	VAR robtarget Openhole_2075 := [[461.97, -18.21, 181.08], [0.041173, 0.705907, 0.7057, -0.044582], [0,0,0,0], [9E9, 9E9, 9E9, 9E9, 9E9, 9E9]];
	VAR robtarget Openhole_2076 := [[462.15, -19.58, 181.25], [0.046371, 0.705585, 0.705943, -0.04055], [0,0,0,0], [9E9, 9E9, 9E9, 9E9, 9E9, 9E9]];
	VAR robtarget Openhole_2077 := [[462.64, -19.54, 181.25], [0.047892, 0.705483, 0.705837, -0.04236], [0,0,0,0], [9E9, 9E9, 9E9, 9E9, 9E9, 9E9]];
	VAR robtarget Openhole_2078 := [[463.64, -19.43, 181.24], [0.050847, 0.705276, 0.705606, -0.046042], [0,0,0,0], [9E9, 9E9, 9E9, 9E9, 9E9, 9E9]];
	VAR robtarget Openhole_2079 := [[464.14, -19.42, 181.24], [0.052483, 0.705156, 0.705494, -0.047735], [0,0,0,0], [9E9, 9E9, 9E9, 9E9, 9E9, 9E9]];
	VAR robtarget Openhole_2080 := [[464.64, -19.38, 181.23], [0.054002, 0.705042, 0.70537, -0.049529], [0,0,0,0], [9E9, 9E9, 9E9, 9E9, 9E9, 9E9]];
	VAR robtarget Openhole_2081 := [[465.63, -19.33, 181.23], [0.05712, 0.704796, 0.705115, -0.053034], [0,0,0,0], [9E9, 9E9, 9E9, 9E9, 9E9, 9E9]];
	VAR robtarget Openhole_2082 := [[466.13, -19.31, 181.23], [0.058717, 0.704665, 0.704985, -0.054743], [0,0,0,0], [9E9, 9E9, 9E9, 9E9, 9E9, 9E9]];
	VAR robtarget Openhole_2083 := [[466.63, -19.31, 181.23], [0.060351, 0.704527, 0.704853, -0.056412], [0,0,0,0], [9E9, 9E9, 9E9, 9E9, 9E9, 9E9]];
	VAR robtarget Openhole_2084 := [[469.13, -19.24, 181.22], [0.068296, 0.703801, 0.704124, -0.064882], [0,0,0,0], [9E9, 9E9, 9E9, 9E9, 9E9, 9E9]];
	VAR robtarget Openhole_2085 := [[469.63, -19.24, 181.22], [0.069931, 0.70364, 0.703972, -0.066512], [0,0,0,0], [9E9, 9E9, 9E9, 9E9, 9E9, 9E9]];
	VAR robtarget Openhole_2086 := [[470.13, -19.24, 181.22], [0.071554, 0.703477, 0.703815, -0.068148], [0,0,0,0], [9E9, 9E9, 9E9, 9E9, 9E9, 9E9]];
	VAR robtarget Openhole_2087 := [[470.63, -19.24, 181.23], [0.073176, 0.70331, 0.703656, -0.069778], [0,0,0,0], [9E9, 9E9, 9E9, 9E9, 9E9, 9E9]];
	VAR robtarget Openhole_2088 := [[490.13, -19.56, 181.39], [0.134065, 0.694281, 0.695212, -0.129154], [0,0,0,0], [9E9, 9E9, 9E9, 9E9, 9E9, 9E9]];
	VAR robtarget Openhole_2089 := [[490.63, -19.56, 181.39], [0.135501, 0.694002, 0.69494, -0.130609], [0,0,0,0], [9E9, 9E9, 9E9, 9E9, 9E9, 9E9]];
	VAR robtarget Openhole_2090 := [[499.63, -19.4, 181.36], [0.159952, 0.688778, 0.689613, -0.156314], [0,0,0,0], [9E9, 9E9, 9E9, 9E9, 9E9, 9E9]];
	VAR robtarget Openhole_2091 := [[504.35, -19.19, 181.27], [0.171684, 0.685948, 0.686508, -0.169431], [0,0,0,0], [9E9, 9E9, 9E9, 9E9, 9E9, 9E9]];
	VAR robtarget Openhole_2092 := [[536.35, -19.19, 181.19], [0.183051, 0.683002, 0.683002, -0.183051], [0,0,0,0], [9E9, 9E9, 9E9, 9E9, 9E9, 9E9]];
	VAR robtarget Openhole_2093 := [[536.35, -19.88, 181.59], [0.183051, 0.683002, 0.683002, -0.183051], [0,0,0,0], [9E9, 9E9, 9E9, 9E9, 9E9, 9E9]];
	VAR robtarget Openhole_2094 := [[509.35, -19.88, 181.68], [0.183051, 0.683002, 0.683002, -0.183051], [0,0,0,0], [9E9, 9E9, 9E9, 9E9, 9E9, 9E9]];
	VAR robtarget Openhole_2095 := [[504.35, -19.88, 181.64], [0.173716, 0.685436, 0.687007, -0.167394], [0,0,0,0], [9E9, 9E9, 9E9, 9E9, 9E9, 9E9]];
	VAR robtarget Openhole_2096 := [[495.85, -20.21, 181.71], [0.152146, 0.690544, 0.692397, -0.14348], [0,0,0,0], [9E9, 9E9, 9E9, 9E9, 9E9, 9E9]];
	VAR robtarget Openhole_2097 := [[489.35, -20.27, 181.66], [0.134036, 0.694287, 0.696036, -0.124637], [0,0,0,0], [9E9, 9E9, 9E9, 9E9, 9E9, 9E9]];
	VAR robtarget Openhole_2098 := [[488.85, -20.27, 181.65], [0.132589, 0.694565, 0.696297, -0.123167], [0,0,0,0], [9E9, 9E9, 9E9, 9E9, 9E9, 9E9]];
	VAR robtarget Openhole_2099 := [[474.85, -20.03, 181.43], [0.089308, 0.701444, 0.702476, -0.080793], [0,0,0,0], [9E9, 9E9, 9E9, 9E9, 9E9, 9E9]];
	VAR robtarget Openhole_2100 := [[470.86, -19.93, 181.37], [0.076174, 0.702992, 0.703809, -0.068212], [0,0,0,0], [9E9, 9E9, 9E9, 9E9, 9E9, 9E9]];
	VAR robtarget Openhole_2101 := [[473.3, -13.93, 180.01], [0.064302, 0.704177, 0.700574, -0.095897], [0,0,0,0], [9E9, 9E9, 9E9, 9E9, 9E9, 9E9]];
	VAR robtarget Openhole_2102 := [[474.29, -13.82, 179.93], [0.067149, 0.703911, 0.700086, -0.099395], [0,0,0,0], [9E9, 9E9, 9E9, 9E9, 9E9, 9E9]];
	VAR robtarget Openhole_2103 := [[479.28, -13.55, 179.6], [0.082192, 0.702314, 0.697567, -0.11576], [0,0,0,0], [9E9, 9E9, 9E9, 9E9, 9E9, 9E9]];
	VAR robtarget Openhole_2104 := [[482.27, -13.53, 179.44], [0.091487, 0.701163, 0.695983, -0.12493], [0,0,0,0], [9E9, 9E9, 9E9, 9E9, 9E9, 9E9]];
	VAR robtarget Openhole_2105 := [[482.77, -13.53, 179.41], [0.093043, 0.700959, 0.695714, -0.12642], [0,0,0,0], [9E9, 9E9, 9E9, 9E9, 9E9, 9E9]];
	VAR robtarget Openhole_2106 := [[494.76, -13.69, 178.85], [0.129253, 0.695193, 0.688701, -0.160282], [0,0,0,0], [9E9, 9E9, 9E9, 9E9, 9E9, 9E9]];
	VAR robtarget Openhole_2107 := [[495.25, -13.69, 178.82], [0.130674, 0.694928, 0.688382, -0.161647], [0,0,0,0], [9E9, 9E9, 9E9, 9E9, 9E9, 9E9]];
	VAR robtarget Openhole_2108 := [[501.74, -13.52, 178.4], [0.148158, 0.691411, 0.683992, -0.179317], [0,0,0,0], [9E9, 9E9, 9E9, 9E9, 9E9, 9E9]];
	VAR robtarget Openhole_2109 := [[504.34, -13.35, 178.17], [0.154616, 0.689996, 0.682093, -0.186411], [0,0,0,0], [9E9, 9E9, 9E9, 9E9, 9E9, 9E9]];
	VAR robtarget Openhole_2110 := [[509.34, -13.35, 177.9], [0.183051, 0.683002, 0.683002, -0.183051], [0,0,0,0], [9E9, 9E9, 9E9, 9E9, 9E9, 9E9]];
	VAR robtarget Openhole_2111 := [[536.34, -13.35, 177.82], [0.183051, 0.683002, 0.683002, -0.183051], [0,0,0,0], [9E9, 9E9, 9E9, 9E9, 9E9, 9E9]];
	VAR robtarget Openhole_2112 := [[536.33, -11.35, 176.66], [0.183051, 0.683002, 0.683002, -0.183051], [0,0,0,0], [9E9, 9E9, 9E9, 9E9, 9E9, 9E9]];
	VAR robtarget Openhole_2113 := [[509.33, -11.35, 176.75], [0.183051, 0.683002, 0.683002, -0.183051], [0,0,0,0], [9E9, 9E9, 9E9, 9E9, 9E9, 9E9]];
	VAR robtarget Openhole_2114 := [[504.33, -11.35, 177.12], [0.148768, 0.69128, 0.68049, -0.192181], [0,0,0,0], [9E9, 9E9, 9E9, 9E9, 9E9, 9E9]];
	VAR robtarget Openhole_2115 := [[503.51, -11.37, 177.19], [0.146636, 0.691735, 0.681083, -0.190069], [0,0,0,0], [9E9, 9E9, 9E9, 9E9, 9E9, 9E9]];
	VAR robtarget Openhole_2116 := [[498.54, -11.56, 177.65], [0.133524, 0.694386, 0.684651, -0.176787], [0,0,0,0], [9E9, 9E9, 9E9, 9E9, 9E9, 9E9]];
	VAR robtarget Openhole_2117 := [[497.54, -11.57, 177.72], [0.130734, 0.694916, 0.685326, -0.174149], [0,0,0,0], [9E9, 9E9, 9E9, 9E9, 9E9, 9E9]];
	VAR robtarget Openhole_2118 := [[497.04, -11.57, 177.76], [0.129318, 0.695181, 0.685659, -0.172833], [0,0,0,0], [9E9, 9E9, 9E9, 9E9, 9E9, 9E9]];
	VAR robtarget Openhole_2119 := [[482.58, -11.27, 178.7], [0.085227, 0.701952, 0.694483, -0.133017], [0,0,0,0], [9E9, 9E9, 9E9, 9E9, 9E9, 9E9]];
	VAR robtarget Openhole_2120 := [[482.08, -11.28, 178.74], [0.083674, 0.702139, 0.694767, -0.131526], [0,0,0,0], [9E9, 9E9, 9E9, 9E9, 9E9, 9E9]];
	VAR robtarget Openhole_2121 := [[477.1, -11.44, 179.15], [0.068397, 0.703791, 0.697543, -0.115903], [0,0,0,0], [9E9, 9E9, 9E9, 9E9, 9E9, 9E9]];
	VAR robtarget Openhole_2122 := [[473.15, -11.89, 179.55], [0.05708, 0.704799, 0.699699, -0.102087], [0,0,0,0], [9E9, 9E9, 9E9, 9E9, 9E9, 9E9]];
	VAR robtarget Openhole_2123 := [[471.68, -12.15, 179.7], [0.053121, 0.705109, 0.70048, -0.096583], [0,0,0,0], [9E9, 9E9, 9E9, 9E9, 9E9, 9E9]];
	VAR robtarget Openhole_2124 := [[471.19, -12.25, 179.76], [0.05186, 0.705202, 0.700737, -0.094695], [0,0,0,0], [9E9, 9E9, 9E9, 9E9, 9E9, 9E9]];
	VAR robtarget Openhole_2125 := [[470.71, -12.36, 179.81], [0.050637, 0.705291, 0.700994, -0.092778], [0,0,0,0], [9E9, 9E9, 9E9, 9E9, 9E9, 9E9]];
	VAR robtarget Openhole_2126 := [[469.27, -12.75, 179.98], [0.047173, 0.705531, 0.70175, -0.086871], [0,0,0,0], [9E9, 9E9, 9E9, 9E9, 9E9, 9E9]];
	VAR robtarget Openhole_2127 := [[468.32, -13.04, 180.09], [0.044997, 0.705674, 0.702239, -0.082831], [0,0,0,0], [9E9, 9E9, 9E9, 9E9, 9E9, 9E9]];
	VAR robtarget Openhole_2128 := [[467.85, -13.2, 180.14], [0.043961, 0.705739, 0.702478, -0.080777], [0,0,0,0], [9E9, 9E9, 9E9, 9E9, 9E9, 9E9]];
	VAR robtarget Openhole_2129 := [[467.38, -13.37, 180.2], [0.042984, 0.705799, 0.702715, -0.078688], [0,0,0,0], [9E9, 9E9, 9E9, 9E9, 9E9, 9E9]];
	VAR robtarget Openhole_2130 := [[466.46, -13.74, 180.31], [0.04115, 0.705908, 0.703177, -0.074444], [0,0,0,0], [9E9, 9E9, 9E9, 9E9, 9E9, 9E9]];
	VAR robtarget Openhole_2131 := [[466, -13.94, 180.37], [0.040305, 0.705957, 0.703402, -0.072286], [0,0,0,0], [9E9, 9E9, 9E9, 9E9, 9E9, 9E9]];
	VAR robtarget Openhole_2132 := [[465.55, -14.15, 180.42], [0.039502, 0.706003, 0.703623, -0.070106], [0,0,0,0], [9E9, 9E9, 9E9, 9E9, 9E9, 9E9]];
	VAR robtarget Openhole_2133 := [[464.66, -14.6, 180.53], [0.03804, 0.706083, 0.70405, -0.065683], [0,0,0,0], [9E9, 9E9, 9E9, 9E9, 9E9, 9E9]];
	VAR robtarget Openhole_2134 := [[463.79, -15.08, 180.63], [0.036763, 0.70615, 0.704455, -0.061184], [0,0,0,0], [9E9, 9E9, 9E9, 9E9, 9E9, 9E9]];
	VAR robtarget Openhole_2135 := [[462.94, -15.6, 180.73], [0.035643, 0.706208, 0.704836, -0.056628], [0,0,0,0], [9E9, 9E9, 9E9, 9E9, 9E9, 9E9]];
	VAR robtarget Openhole_2136 := [[462.52, -15.87, 180.78], [0.03514, 0.706233, 0.705017, -0.054329], [0,0,0,0], [9E9, 9E9, 9E9, 9E9, 9E9, 9E9]];
	VAR robtarget Openhole_2137 := [[460.89, -17, 180.96], [0.033479, 0.706314, 0.705672, -0.045027], [0,0,0,0], [9E9, 9E9, 9E9, 9E9, 9E9, 9E9]];
	VAR robtarget Openhole_2138 := [[461.06, -13.27, 180.53], [0.021493, 0.70678, 0.704709, -0.058177], [0,0,0,0], [9E9, 9E9, 9E9, 9E9, 9E9, 9E9]];
	VAR robtarget Openhole_2139 := [[460.62, -13.5, 180.58], [0.020785, 0.706801, 0.704891, -0.055928], [0,0,0,0], [9E9, 9E9, 9E9, 9E9, 9E9, 9E9]];
	VAR robtarget Openhole_2140 := [[458.51, -14.82, 180.81], [0.018075, 0.706876, 0.705711, -0.04441], [0,0,0,0], [9E9, 9E9, 9E9, 9E9, 9E9, 9E9]];
	VAR robtarget Openhole_2141 := [[457.68, -15.38, 180.89], [0.017191, 0.706898, 0.705989, -0.039736], [0,0,0,0], [9E9, 9E9, 9E9, 9E9, 9E9, 9E9]];
	VAR robtarget Openhole_2142 := [[456.81, -15.81, 180.95], [0.01568, 0.706933, 0.706224, -0.035314], [0,0,0,0], [9E9, 9E9, 9E9, 9E9, 9E9, 9E9]];
	VAR robtarget Openhole_2143 := [[457.02, -21.12, 181.34], [0.034402, 0.706269, 0.706877, -0.018011], [0,0,0,0], [9E9, 9E9, 9E9, 9E9, 9E9, 9E9]];
	VAR robtarget Openhole_2144 := [[463.92, -21.12, 181.48], [0.057484, 0.704766, 0.7059, -0.041297], [0,0,0,0], [9E9, 9E9, 9E9, 9E9, 9E9, 9E9]];
	VAR robtarget Openhole_2145 := [[469.41, -21.53, 181.67], [0.076804, 0.702923, 0.704714, -0.05812], [0,0,0,0], [9E9, 9E9, 9E9, 9E9, 9E9, 9E9]];
	VAR robtarget Openhole_2146 := [[482.39, -21.87, 182.08], [0.118549, 0.697098, 0.700201, -0.098586], [0,0,0,0], [9E9, 9E9, 9E9, 9E9, 9E9, 9E9]];
	VAR robtarget Openhole_2147 := [[487.39, -21.9, 182.23], [0.133435, 0.694403, 0.697902, -0.113721], [0,0,0,0], [9E9, 9E9, 9E9, 9E9, 9E9, 9E9]];
	VAR robtarget Openhole_2148 := [[487.89, -21.9, 182.25], [0.134884, 0.694123, 0.697657, -0.115218], [0,0,0,0], [9E9, 9E9, 9E9, 9E9, 9E9, 9E9]];
	VAR robtarget Openhole_2149 := [[498.39, -21.73, 182.46], [0.16361, 0.687918, 0.691889, -0.14591], [0,0,0,0], [9E9, 9E9, 9E9, 9E9, 9E9, 9E9]];
	VAR robtarget Openhole_2150 := [[503.38, -21.52, 182.48], [0.176032, 0.684845, 0.688756, -0.160046], [0,0,0,0], [9E9, 9E9, 9E9, 9E9, 9E9, 9E9]];
	VAR robtarget Openhole_2151 := [[504.35, -21.49, 182.49], [0.178402, 0.684232, 0.688137, -0.162688], [0,0,0,0], [9E9, 9E9, 9E9, 9E9, 9E9, 9E9]];
	VAR robtarget Openhole_2152 := [[509.35, -21.49, 182.61], [0.183051, 0.683002, 0.683002, -0.183051], [0,0,0,0], [9E9, 9E9, 9E9, 9E9, 9E9, 9E9]];
	VAR robtarget Openhole_2153 := [[536.24, -21.49, 182.52], [0.183051, 0.683002, 0.683002, -0.183051], [0,0,0,0], [9E9, 9E9, 9E9, 9E9, 9E9, 9E9]];
	VAR robtarget Openhole_2154 := [[536.33, -31.04, 188.04], [0.183051, 0.683002, 0.683002, -0.183051], [0,0,0,0], [9E9, 9E9, 9E9, 9E9, 9E9, 9E9]];
	VAR robtarget Openhole_2155 := [[509.37, -31.04, 188.12], [0.183051, 0.683002, 0.683002, -0.183051], [0,0,0,0], [9E9, 9E9, 9E9, 9E9, 9E9, 9E9]];
	VAR robtarget Openhole_2156 := [[504.38, -31.04, 187.54], [0.205934, 0.676455, 0.694141, -0.134788], [0,0,0,0], [9E9, 9E9, 9E9, 9E9, 9E9, 9E9]];
	VAR robtarget Openhole_2157 := [[486.98, -32.16, 185.94], [0.164078, 0.687807, 0.702555, -0.080102], [0,0,0,0], [9E9, 9E9, 9E9, 9E9, 9E9, 9E9]];
	VAR robtarget Openhole_2158 := [[478.56, -33.01, 185.11], [0.142475, 0.692604, 0.705303, -0.050481], [0,0,0,0], [9E9, 9E9, 9E9, 9E9, 9E9, 9E9]];
	VAR robtarget Openhole_2159 := [[471.67, -34.05, 184.41], [0.124885, 0.695991, 0.706689, -0.024306], [0,0,0,0], [9E9, 9E9, 9E9, 9E9, 9E9, 9E9]];
	VAR robtarget Openhole_2160 := [[465.83, -35.24, 183.75], [0.110356, 0.698442, 0.707106, -0.000639], [0,0,0,0], [9E9, 9E9, 9E9, 9E9, 9E9, 9E9]];
	VAR robtarget Openhole_2161 := [[458.15, -37.22, 182.72], [0.091834, 0.701118, 0.706377, 0.032124], [0,0,0,0], [9E9, 9E9, 9E9, 9E9, 9E9, 9E9]];
	VAR robtarget Openhole_2162 := [[452.92, -38.7, 181.86], [0.079284, 0.702648, 0.704975, 0.054868], [0,0,0,0], [9E9, 9E9, 9E9, 9E9, 9E9, 9E9]];
	VAR robtarget Openhole_2163 := [[457.28, -38.7, 182.68], [0.093765, 0.700862, 0.705976, 0.039977], [0,0,0,0], [9E9, 9E9, 9E9, 9E9, 9E9, 9E9]];
	VAR robtarget Openhole_2164 := [[457.75, -38.56, 182.76], [0.094884, 0.700712, 0.706092, 0.037872], [0,0,0,0], [9E9, 9E9, 9E9, 9E9, 9E9, 9E9]];
	VAR robtarget Openhole_2165 := [[466.4, -36.39, 184.03], [0.115866, 0.697549, 0.707106, 0.001208], [0,0,0,0], [9E9, 9E9, 9E9, 9E9, 9E9, 9E9]];
	VAR robtarget Openhole_2166 := [[473.19, -34.93, 184.83], [0.132384, 0.694604, 0.706609, -0.026523], [0,0,0,0], [9E9, 9E9, 9E9, 9E9, 9E9, 9E9]];
	VAR robtarget Openhole_2167 := [[479.58, -33.93, 185.52], [0.148359, 0.691368, 0.705275, -0.050864], [0,0,0,0], [9E9, 9E9, 9E9, 9E9, 9E9, 9E9]];
	VAR robtarget Openhole_2168 := [[487.99, -33.03, 186.39], [0.169538, 0.686482, 0.702507, -0.080521], [0,0,0,0], [9E9, 9E9, 9E9, 9E9, 9E9, 9E9]];
	VAR robtarget Openhole_2169 := [[504.38, -31.93, 188.01], [0.208432, 0.675689, 0.69464, -0.132194], [0,0,0,0], [9E9, 9E9, 9E9, 9E9, 9E9, 9E9]];
	VAR robtarget Openhole_2170 := [[509.37, -31.93, 188.63], [0.183051, 0.683002, 0.683002, -0.183051], [0,0,0,0], [9E9, 9E9, 9E9, 9E9, 9E9, 9E9]];
	VAR robtarget Openhole_2171 := [[536.37, -31.93, 188.55], [0.183051, 0.683002, 0.683002, -0.183051], [0,0,0,0], [9E9, 9E9, 9E9, 9E9, 9E9, 9E9]];
	VAR robtarget Openhole_2172 := [[536.37, -32.81, 189.06], [0.183051, 0.683002, 0.683002, -0.183051], [0,0,0,0], [9E9, 9E9, 9E9, 9E9, 9E9, 9E9]];
	VAR robtarget Openhole_2173 := [[524.37, -32.81, 189.09], [0.183051, 0.683002, 0.683002, -0.183051], [0,0,0,0], [9E9, 9E9, 9E9, 9E9, 9E9, 9E9]];
	VAR robtarget Openhole_2174 := [[509.37, -32.81, 189.14], [0.183051, 0.683002, 0.683002, -0.183051], [0,0,0,0], [9E9, 9E9, 9E9, 9E9, 9E9, 9E9]];
	VAR robtarget Openhole_2175 := [[504.38, -32.81, 188.48], [0.210931, 0.674914, 0.695127, -0.12961], [0,0,0,0], [9E9, 9E9, 9E9, 9E9, 9E9, 9E9]];
	VAR robtarget Openhole_2176 := [[488.99, -33.88, 186.85], [0.17487, 0.685143, 0.702451, -0.081013], [0,0,0,0], [9E9, 9E9, 9E9, 9E9, 9E9, 9E9]];
	VAR robtarget Openhole_2177 := [[481.09, -34.74, 185.98], [0.155283, 0.689846, 0.705104, -0.053183], [0,0,0,0], [9E9, 9E9, 9E9, 9E9, 9E9, 9E9]];
	VAR robtarget Openhole_2178 := [[474.71, -35.76, 185.26], [0.139596, 0.69319, 0.706515, -0.028917], [0,0,0,0], [9E9, 9E9, 9E9, 9E9, 9E9, 9E9]];
	VAR robtarget Openhole_2179 := [[467.43, -37.31, 184.36], [0.122079, 0.696489, 0.707106, 0.000696], [0,0,0,0], [9E9, 9E9, 9E9, 9E9, 9E9, 9E9]];
	VAR robtarget Openhole_2180 := [[462.62, -38.48, 183.66], [0.110468, 0.698425, 0.706797, 0.020931], [0,0,0,0], [9E9, 9E9, 9E9, 9E9, 9E9, 9E9]];
	VAR robtarget Openhole_2181 := [[462.13, -38.7, 183.6], [0.109631, 0.698556, 0.706722, 0.023316], [0,0,0,0], [9E9, 9E9, 9E9, 9E9, 9E9, 9E9]];
	VAR robtarget Openhole_2182 := [[466.52, -38.7, 184.43], [0.123628, 0.696216, 0.707058, 0.00831], [0,0,0,0], [9E9, 9E9, 9E9, 9E9, 9E9, 9E9]];
	VAR robtarget Openhole_2183 := [[467, -38.47, 184.48], [0.124426, 0.696073, 0.707082, 0.00591], [0,0,0,0], [9E9, 9E9, 9E9, 9E9, 9E9, 9E9]];
	VAR robtarget Openhole_2184 := [[474.26, -36.86, 185.46], [0.141738, 0.692756, 0.706704, -0.023852], [0,0,0,0], [9E9, 9E9, 9E9, 9E9, 9E9, 9E9]];
	VAR robtarget Openhole_2185 := [[481.12, -35.71, 186.28], [0.158391, 0.689139, 0.705324, -0.050174], [0,0,0,0], [9E9, 9E9, 9E9, 9E9, 9E9, 9E9]];
	VAR robtarget Openhole_2186 := [[489.01, -34.8, 187.2], [0.177697, 0.684415, 0.702769, -0.078203], [0,0,0,0], [9E9, 9E9, 9E9, 9E9, 9E9, 9E9]];
	VAR robtarget Openhole_2187 := [[501.89, -33.86, 188.68], [0.207948, 0.675838, 0.696929, -0.119541], [0,0,0,0], [9E9, 9E9, 9E9, 9E9, 9E9, 9E9]];
	VAR robtarget Openhole_2188 := [[504.38, -33.69, 188.95], [0.213421, 0.67413, 0.695603, -0.127028], [0,0,0,0], [9E9, 9E9, 9E9, 9E9, 9E9, 9E9]];
	VAR robtarget Openhole_2189 := [[509.37, -33.69, 189.65], [0.183051, 0.683002, 0.683002, -0.183051], [0,0,0,0], [9E9, 9E9, 9E9, 9E9, 9E9, 9E9]];
	VAR robtarget Openhole_2190 := [[536.37, -33.69, 189.57], [0.183051, 0.683002, 0.683002, -0.183051], [0,0,0,0], [9E9, 9E9, 9E9, 9E9, 9E9, 9E9]];
	VAR robtarget Openhole_2191 := [[536.37, -34.58, 190.08], [0.183051, 0.683002, 0.683002, -0.183051], [0,0,0,0], [9E9, 9E9, 9E9, 9E9, 9E9, 9E9]];
	VAR robtarget Openhole_2192 := [[509.37, -34.58, 190.16], [0.183051, 0.683002, 0.683002, -0.183051], [0,0,0,0], [9E9, 9E9, 9E9, 9E9, 9E9, 9E9]];
	VAR robtarget Openhole_2193 := [[504.37, -34.58, 189.41], [0.2159, 0.67334, 0.696071, -0.124442], [0,0,0,0], [9E9, 9E9, 9E9, 9E9, 9E9, 9E9]];
	VAR robtarget Openhole_2194 := [[490.51, -35.57, 187.73], [0.184036, 0.682738, 0.702511, -0.080486], [0,0,0,0], [9E9, 9E9, 9E9, 9E9, 9E9, 9E9]];
	VAR robtarget Openhole_2195 := [[482.13, -36.52, 186.7], [0.163758, 0.687883, 0.705271, -0.050922], [0,0,0,0], [9E9, 9E9, 9E9, 9E9, 9E9, 9E9]];
	VAR robtarget Openhole_2196 := [[475.27, -37.64, 185.82], [0.147219, 0.691611, 0.706674, -0.024743], [0,0,0,0], [9E9, 9E9, 9E9, 9E9, 9E9, 9E9]];
	VAR robtarget Openhole_2197 := [[470.91, -38.55, 185.23], [0.136836, 0.693741, 0.707071, -0.007115], [0,0,0,0], [9E9, 9E9, 9E9, 9E9, 9E9, 9E9]];
	VAR robtarget Openhole_2198 := [[470.42, -38.7, 185.17], [0.135813, 0.693942, 0.707089, -0.004993], [0,0,0,0], [9E9, 9E9, 9E9, 9E9, 9E9, 9E9]];
	VAR robtarget Openhole_2199 := [[474.82, -38.7, 186], [0.149173, 0.691193, 0.706828, -0.019841], [0,0,0,0], [9E9, 9E9, 9E9, 9E9, 9E9, 9E9]];
	VAR robtarget Openhole_2200 := [[475.31, -38.59, 186.07], [0.150274, 0.690954, 0.706769, -0.021839], [0,0,0,0], [9E9, 9E9, 9E9, 9E9, 9E9, 9E9]];
	VAR robtarget Openhole_2201 := [[482.64, -37.38, 187.06], [0.167864, 0.686893, 0.705345, -0.049885], [0,0,0,0], [9E9, 9E9, 9E9, 9E9, 9E9, 9E9]];
	VAR robtarget Openhole_2202 := [[491.02, -36.43, 188.16], [0.187921, 0.681679, 0.70263, -0.07944], [0,0,0,0], [9E9, 9E9, 9E9, 9E9, 9E9, 9E9]];
	VAR robtarget Openhole_2203 := [[502.39, -35.58, 189.63], [0.214044, 0.673933, 0.697545, -0.115895], [0,0,0,0], [9E9, 9E9, 9E9, 9E9, 9E9, 9E9]];
	VAR robtarget Openhole_2204 := [[504.37, -35.46, 189.88], [0.218376, 0.672541, 0.696526, -0.121866], [0,0,0,0], [9E9, 9E9, 9E9, 9E9, 9E9, 9E9]];
	VAR robtarget Openhole_2205 := [[504.37, -35.46, 189.88], [0.21838, 0.67254, 0.696525, -0.121873], [0,0,0,0], [9E9, 9E9, 9E9, 9E9, 9E9, 9E9]];
	VAR robtarget Openhole_2206 := [[509.38, -35.46, 190.67], [0.183051, 0.683002, 0.683002, -0.183051], [0,0,0,0], [9E9, 9E9, 9E9, 9E9, 9E9, 9E9]];
	VAR robtarget Openhole_2207 := [[536.38, -35.46, 190.59], [0.183051, 0.683002, 0.683002, -0.183051], [0,0,0,0], [9E9, 9E9, 9E9, 9E9, 9E9, 9E9]];
	VAR robtarget Openhole_2208 := [[536.38, -36.35, 191.1], [0.183051, 0.683002, 0.683002, -0.183051], [0,0,0,0], [9E9, 9E9, 9E9, 9E9, 9E9, 9E9]];
	VAR robtarget Openhole_2209 := [[509.38, -36.35, 191.18], [0.183051, 0.683002, 0.683002, -0.183051], [0,0,0,0], [9E9, 9E9, 9E9, 9E9, 9E9, 9E9]];
	VAR robtarget Openhole_2210 := [[504.37, -36.35, 190.35], [0.220853, 0.671732, 0.696969, -0.119308], [0,0,0,0], [9E9, 9E9, 9E9, 9E9, 9E9, 9E9]];
	VAR robtarget Openhole_2211 := [[504.37, -36.35, 190.35], [0.220841, 0.671736, 0.696972, -0.119291], [0,0,0,0], [9E9, 9E9, 9E9, 9E9, 9E9, 9E9]];
	VAR robtarget Openhole_2212 := [[503.87, -36.37, 190.28], [0.219768, 0.672088, 0.697224, -0.117808], [0,0,0,0], [9E9, 9E9, 9E9, 9E9, 9E9, 9E9]];
	VAR robtarget Openhole_2213 := [[492.02, -37.26, 188.67], [0.193013, 0.680254, 0.702569, -0.079982], [0,0,0,0], [9E9, 9E9, 9E9, 9E9, 9E9, 9E9]];
	VAR robtarget Openhole_2214 := [[483.16, -38.26, 187.44], [0.172017, 0.685865, 0.705422, -0.04878], [0,0,0,0], [9E9, 9E9, 9E9, 9E9, 9E9, 9E9]];
	VAR robtarget Openhole_2215 := [[480.22, -38.7, 187.02], [0.165, 0.687586, 0.706096, -0.037791], [0,0,0,0], [9E9, 9E9, 9E9, 9E9, 9E9, 9E9]];
	VAR robtarget Openhole_2216 := [[389.31, -38.7, 169.82], [-0.12615, 0.695763, 0.665642, 0.238581], [0,0,0,0], [9E9, 9E9, 9E9, 9E9, 9E9, 9E9]];
	VAR robtarget Openhole_2217 := [[361.4, -38.7, 169.91], [-0.183051, 0.683002, 0.683002, 0.183051], [0,0,0,0], [9E9, 9E9, 9E9, 9E9, 9E9, 9E9]];
	VAR robtarget Openhole_2218 := [[362.33, -29.87, 175], [-0.183051, 0.683002, 0.683002, 0.183051], [0,0,0,0], [9E9, 9E9, 9E9, 9E9, 9E9, 9E9]];
	VAR robtarget Openhole_2219 := [[389.33, -29.87, 174.92], [-0.1512, 0.690752, 0.673839, 0.214338], [0,0,0,0], [9E9, 9E9, 9E9, 9E9, 9E9, 9E9]];
	VAR robtarget Openhole_2220 := [[394.33, -29.87, 175.44], [-0.137763, 0.693557, 0.677476, 0.202551], [0,0,0,0], [9E9, 9E9, 9E9, 9E9, 9E9, 9E9]];
	VAR robtarget Openhole_2221 := [[394.88, -29.88, 175.49], [-0.136237, 0.693858, 0.677866, 0.20124], [0,0,0,0], [9E9, 9E9, 9E9, 9E9, 9E9, 9E9]];
	VAR robtarget Openhole_2222 := [[399.85, -30.07, 175.92], [-0.121699, 0.696555, 0.681266, 0.18941], [0,0,0,0], [9E9, 9E9, 9E9, 9E9, 9E9, 9E9]];
	VAR robtarget Openhole_2223 := [[412.28, -31.06, 176.89], [-0.081421, 0.702403, 0.688984, 0.159062], [0,0,0,0], [9E9, 9E9, 9E9, 9E9, 9E9, 9E9]];
	VAR robtarget Openhole_2224 := [[418.24, -31.27, 177.52], [-0.061858, 0.704396, 0.692601, 0.142491], [0,0,0,0], [9E9, 9E9, 9E9, 9E9, 9E9, 9E9]];
	VAR robtarget Openhole_2225 := [[418.73, -31.27, 177.58], [-0.06026, 0.704534, 0.692902, 0.141019], [0,0,0,0], [9E9, 9E9, 9E9, 9E9, 9E9, 9E9]];
	VAR robtarget Openhole_2226 := [[423.69, -31.07, 178.21], [-0.044741, 0.70569, 0.695888, 0.125456], [0,0,0,0], [9E9, 9E9, 9E9, 9E9, 9E9, 9E9]];
	VAR robtarget Openhole_2227 := [[428.61, -30.5, 178.89], [-0.030265, 0.706459, 0.698762, 0.10831], [0,0,0,0], [9E9, 9E9, 9E9, 9E9, 9E9, 9E9]];
	VAR robtarget Openhole_2228 := [[434.94, -29.34, 179.75], [-0.012795, 0.706991, 0.702086, 0.084111], [0,0,0,0], [9E9, 9E9, 9E9, 9E9, 9E9, 9E9]];
	VAR robtarget Openhole_2229 := [[437.87, -28.76, 180.11], [-0.004847, 0.70709, 0.703374, 0.07256], [0,0,0,0], [9E9, 9E9, 9E9, 9E9, 9E9, 9E9]];
	VAR robtarget Openhole_2230 := [[438.84, -28.58, 180.22], [-0.002113, 0.707104, 0.703759, 0.06873], [0,0,0,0], [9E9, 9E9, 9E9, 9E9, 9E9, 9E9]];
	VAR robtarget Openhole_2231 := [[441.3, -28.17, 180.47], [0.00485, 0.70709, 0.704626, 0.059176], [0,0,0,0], [9E9, 9E9, 9E9, 9E9, 9E9, 9E9]];
	VAR robtarget Openhole_2232 := [[442.28, -28.03, 180.57], [0.007732, 0.707065, 0.704933, 0.055401], [0,0,0,0], [9E9, 9E9, 9E9, 9E9, 9E9, 9E9]];
	VAR robtarget Openhole_2233 := [[445.74, -27.57, 180.88], [0.017944, 0.706879, 0.705846, 0.0422], [0,0,0,0], [9E9, 9E9, 9E9, 9E9, 9E9, 9E9]];
	VAR robtarget Openhole_2234 := [[447.22, -27.43, 181.01], [0.022536, 0.706748, 0.706155, 0.036685], [0,0,0,0], [9E9, 9E9, 9E9, 9E9, 9E9, 9E9]];
	VAR robtarget Openhole_2235 := [[447.72, -27.4, 181.05], [0.02415, 0.706694, 0.706244, 0.034916], [0,0,0,0], [9E9, 9E9, 9E9, 9E9, 9E9, 9E9]];
	VAR robtarget Openhole_2236 := [[448.22, -27.39, 181.09], [0.025802, 0.706636, 0.706328, 0.033182], [0,0,0,0], [9E9, 9E9, 9E9, 9E9, 9E9, 9E9]];
	VAR robtarget Openhole_2237 := [[448.72, -27.39, 181.13], [0.027502, 0.706572, 0.706405, 0.031494], [0,0,0,0], [9E9, 9E9, 9E9, 9E9, 9E9, 9E9]];
	VAR robtarget Openhole_2238 := [[452.7, -27.62, 181.46], [0.041775, 0.705872, 0.706859, 0.018727], [0,0,0,0], [9E9, 9E9, 9E9, 9E9, 9E9, 9E9]];
	VAR robtarget Openhole_2239 := [[454.19, -27.71, 181.59], [0.047103, 0.705536, 0.70697, 0.013931], [0,0,0,0], [9E9, 9E9, 9E9, 9E9, 9E9, 9E9]];
	VAR robtarget Openhole_2240 := [[454.69, -27.73, 181.63], [0.048848, 0.705418, 0.707, 0.012303], [0,0,0,0], [9E9, 9E9, 9E9, 9E9, 9E9, 9E9]];
	VAR robtarget Openhole_2241 := [[455.68, -27.74, 181.71], [0.052246, 0.705174, 0.70705, 0.008952], [0,0,0,0], [9E9, 9E9, 9E9, 9E9, 9E9, 9E9]];
	VAR robtarget Openhole_2242 := [[456.18, -27.73, 181.75], [0.053883, 0.705051, 0.70707, 0.007217], [0,0,0,0], [9E9, 9E9, 9E9, 9E9, 9E9, 9E9]];
	VAR robtarget Openhole_2243 := [[473.12, -27.13, 183.03], [0.107027, 0.69896, 0.705205, -0.051819], [0,0,0,0], [9E9, 9E9, 9E9, 9E9, 9E9, 9E9]];
	VAR robtarget Openhole_2244 := [[498.06, -26.27, 184.58], [0.176241, 0.684791, 0.694806, -0.131317], [0,0,0,0], [9E9, 9E9, 9E9, 9E9, 9E9, 9E9]];
	VAR robtarget Openhole_2245 := [[504.36, -25.98, 184.86], [0.191383, 0.680715, 0.691107, -0.149567], [0,0,0,0], [9E9, 9E9, 9E9, 9E9, 9E9, 9E9]];
	VAR robtarget Openhole_2246 := [[509.36, -25.98, 185.19], [0.183051, 0.683002, 0.683002, -0.183051], [0,0,0,0], [9E9, 9E9, 9E9, 9E9, 9E9, 9E9]];
	VAR robtarget Openhole_2247 := [[536.36, -25.98, 185.11], [0.183051, 0.683002, 0.683002, -0.183051], [0,0,0,0], [9E9, 9E9, 9E9, 9E9, 9E9, 9E9]];
	VAR robtarget Openhole_2248 := [[536.36, -24.92, 184.5], [0.183051, 0.683002, 0.683002, -0.183051], [0,0,0,0], [9E9, 9E9, 9E9, 9E9, 9E9, 9E9]];
	VAR robtarget Openhole_2249 := [[509.36, -24.92, 184.58], [0.183051, 0.683002, 0.683002, -0.183051], [0,0,0,0], [9E9, 9E9, 9E9, 9E9, 9E9, 9E9]];
	VAR robtarget Openhole_2250 := [[504.36, -24.92, 184.3], [0.188332, 0.681565, 0.690431, -0.152662], [0,0,0,0], [9E9, 9E9, 9E9, 9E9, 9E9, 9E9]];
	VAR robtarget Openhole_2251 := [[493.09, -25.36, 183.85], [0.160233, 0.688713, 0.696886, -0.119791], [0,0,0,0], [9E9, 9E9, 9E9, 9E9, 9E9, 9E9]];
	VAR robtarget Openhole_2252 := [[469.64, -25.84, 182.51], [0.091778, 0.701125, 0.705702, -0.044555], [0,0,0,0], [9E9, 9E9, 9E9, 9E9, 9E9, 9E9]];
	VAR robtarget Openhole_2253 := [[467.64, -25.85, 182.38], [0.085401, 0.701931, 0.706092, -0.037869], [0,0,0,0], [9E9, 9E9, 9E9, 9E9, 9E9, 9E9]];
	VAR robtarget Openhole_2254 := [[467.14, -25.85, 182.35], [0.083781, 0.702126, 0.706179, -0.036207], [0,0,0,0], [9E9, 9E9, 9E9, 9E9, 9E9, 9E9]];
	VAR robtarget Openhole_2255 := [[459.66, -25.63, 181.84], [0.058467, 0.704685, 0.70701, -0.011719], [0,0,0,0], [9E9, 9E9, 9E9, 9E9, 9E9, 9E9]];
	VAR robtarget Openhole_2256 := [[455.68, -25.42, 181.57], [0.044398, 0.705712, 0.707106, 0.001113], [0,0,0,0], [9E9, 9E9, 9E9, 9E9, 9E9, 9E9]];
	VAR robtarget Openhole_2257 := [[455.18, -25.38, 181.54], [0.042578, 0.705824, 0.707102, 0.002659], [0,0,0,0], [9E9, 9E9, 9E9, 9E9, 9E9, 9E9]];
	VAR robtarget Openhole_2258 := [[454.68, -25.32, 181.5], [0.040725, 0.705933, 0.707094, 0.004169], [0,0,0,0], [9E9, 9E9, 9E9, 9E9, 9E9, 9E9]];
	VAR robtarget Openhole_2259 := [[454.1, -25.14, 181.46], [0.038116, 0.706079, 0.707085, 0.005549], [0,0,0,0], [9E9, 9E9, 9E9, 9E9, 9E9, 9E9]];
	VAR robtarget Openhole_2260 := [[451.65, -25.14, 181.32], [0.029833, 0.706477, 0.70697, 0.013891], [0,0,0,0], [9E9, 9E9, 9E9, 9E9, 9E9, 9E9]];
	VAR robtarget Openhole_2261 := [[453.07, -23.79, 181.35], [0.030088, 0.706466, 0.707093, 0.004445], [0,0,0,0], [9E9, 9E9, 9E9, 9E9, 9E9, 9E9]];
	VAR robtarget Openhole_2262 := [[455.52, -23.79, 181.46], [0.038358, 0.706066, 0.707096, -0.00389], [0,0,0,0], [9E9, 9E9, 9E9, 9E9, 9E9, 9E9]];
	VAR robtarget Openhole_2263 := [[456.08, -23.86, 181.49], [0.040496, 0.705946, 0.707085, -0.005547], [0,0,0,0], [9E9, 9E9, 9E9, 9E9, 9E9, 9E9]];
	VAR robtarget Openhole_2264 := [[457.08, -23.91, 181.54], [0.044021, 0.705735, 0.707052, -0.00877], [0,0,0,0], [9E9, 9E9, 9E9, 9E9, 9E9, 9E9]];
	VAR robtarget Openhole_2265 := [[458.58, -23.97, 181.62], [0.049247, 0.70539, 0.706975, -0.013649], [0,0,0,0], [9E9, 9E9, 9E9, 9E9, 9E9, 9E9]];
	VAR robtarget Openhole_2266 := [[465.04, -24.53, 182.01], [0.072538, 0.703376, 0.706308, -0.033597], [0,0,0,0], [9E9, 9E9, 9E9, 9E9, 9E9, 9E9]];
	VAR robtarget Openhole_2267 := [[473.02, -24.68, 182.47], [0.098727, 0.700181, 0.704593, -0.059575], [0,0,0,0], [9E9, 9E9, 9E9, 9E9, 9E9, 9E9]];
	VAR robtarget Openhole_2268 := [[473.52, -24.68, 182.5], [0.1003, 0.699957, 0.704453, -0.061206], [0,0,0,0], [9E9, 9E9, 9E9, 9E9, 9E9, 9E9]];
	VAR robtarget Openhole_2269 := [[491, -24.49, 183.37], [0.151774, 0.690626, 0.69747, -0.116343], [0,0,0,0], [9E9, 9E9, 9E9, 9E9, 9E9, 9E9]];
	VAR robtarget Openhole_2270 := [[501.99, -24.14, 183.77], [0.180115, 0.683782, 0.691322, -0.148574], [0,0,0,0], [9E9, 9E9, 9E9, 9E9, 9E9, 9E9]];
	VAR robtarget Openhole_2271 := [[504.35, -24.03, 183.83], [0.185766, 0.682269, 0.689851, -0.15526], [0,0,0,0], [9E9, 9E9, 9E9, 9E9, 9E9, 9E9]];
	VAR robtarget Openhole_2272 := [[509.36, -24.03, 184.07], [0.183051, 0.683002, 0.683002, -0.183051], [0,0,0,0], [9E9, 9E9, 9E9, 9E9, 9E9, 9E9]];
	VAR robtarget Openhole_2273 := [[536.36, -24.03, 183.99], [0.183051, 0.683002, 0.683002, -0.183051], [0,0,0,0], [9E9, 9E9, 9E9, 9E9, 9E9, 9E9]];
	VAR robtarget Openhole_2274 := [[536.35, -23.14, 183.47], [0.183051, 0.683002, 0.683002, -0.183051], [0,0,0,0], [9E9, 9E9, 9E9, 9E9, 9E9, 9E9]];
	VAR robtarget Openhole_2275 := [[509.35, -23.14, 183.56], [0.183051, 0.683002, 0.683002, -0.183051], [0,0,0,0], [9E9, 9E9, 9E9, 9E9, 9E9, 9E9]];
	VAR robtarget Openhole_2276 := [[504.35, -23.14, 183.36], [0.183175, 0.682969, 0.689256, -0.157878], [0,0,0,0], [9E9, 9E9, 9E9, 9E9, 9E9, 9E9]];
	VAR robtarget Openhole_2277 := [[494.81, -23.51, 183.14], [0.159285, 0.688933, 0.694968, -0.130461], [0,0,0,0], [9E9, 9E9, 9E9, 9E9, 9E9, 9E9]];
	VAR robtarget Openhole_2278 := [[481.32, -23.66, 182.61], [0.121032, 0.696672, 0.701423, -0.089474], [0,0,0,0], [9E9, 9E9, 9E9, 9E9, 9E9, 9E9]];
	VAR robtarget Openhole_2279 := [[480.82, -23.66, 182.58], [0.119525, 0.696932, 0.701621, -0.087907], [0,0,0,0], [9E9, 9E9, 9E9, 9E9, 9E9, 9E9]];
	VAR robtarget Openhole_2280 := [[480.32, -23.66, 182.56], [0.118013, 0.697189, 0.701816, -0.086336], [0,0,0,0], [9E9, 9E9, 9E9, 9E9, 9E9, 9E9]];
	VAR robtarget Openhole_2281 := [[479.82, -23.66, 182.54], [0.116493, 0.697445, 0.702008, -0.084763], [0,0,0,0], [9E9, 9E9, 9E9, 9E9, 9E9, 9E9]];
	VAR robtarget Openhole_2282 := [[468.84, -23.5, 182.02], [0.081465, 0.702398, 0.705358, -0.049695], [0,0,0,0], [9E9, 9E9, 9E9, 9E9, 9E9, 9E9]];
	VAR robtarget Openhole_2283 := [[463.85, -23.16, 181.76], [0.064065, 0.704199, 0.706278, -0.034217], [0,0,0,0], [9E9, 9E9, 9E9, 9E9, 9E9, 9E9]];
	VAR robtarget Openhole_2284 := [[459.89, -22.67, 181.55], [0.049272, 0.705388, 0.706749, -0.022481], [0,0,0,0], [9E9, 9E9, 9E9, 9E9, 9E9, 9E9]];
	VAR robtarget Openhole_2285 := [[458.89, -22.62, 181.51], [0.045756, 0.705625, 0.706844, -0.019279], [0,0,0,0], [9E9, 9E9, 9E9, 9E9, 9E9, 9E9]];
	VAR robtarget Openhole_2286 := [[457.39, -22.58, 181.46], [0.040573, 0.705942, 0.706961, -0.014351], [0,0,0,0], [9E9, 9E9, 9E9, 9E9, 9E9, 9E9]];
	VAR robtarget Openhole_2287 := [[456.89, -22.57, 181.44], [0.038877, 0.706037, 0.706993, -0.012669], [0,0,0,0], [9E9, 9E9, 9E9, 9E9, 9E9, 9E9]];
	VAR robtarget Openhole_2288 := [[456.36, -22.56, 181.42], [0.037011, 0.706138, 0.707023, -0.010896], [0,0,0,0], [9E9, 9E9, 9E9, 9E9, 9E9, 9E9]];
	VAR robtarget Openhole_2289 := [[453.91, -22.56, 181.34], [0.028745, 0.706522, 0.707102, -0.002569], [0,0,0,0], [9E9, 9E9, 9E9, 9E9, 9E9, 9E9]];
	VAR robtarget Openhole_2290 := [[454.35, -21.6, 181.31], [0.027022, 0.70659, 0.707069, -0.007322], [0,0,0,0], [9E9, 9E9, 9E9, 9E9, 9E9, 9E9]];
	VAR robtarget Openhole_2291 := [[456.8, -21.6, 181.37], [0.035288, 0.706226, 0.706934, -0.01564], [0,0,0,0], [9E9, 9E9, 9E9, 9E9, 9E9, 9E9]];
	VAR robtarget Openhole_2292 := [[457.66, -21.63, 181.39], [0.038264, 0.706071, 0.706866, -0.018465], [0,0,0,0], [9E9, 9E9, 9E9, 9E9, 9E9, 9E9]];
	VAR robtarget Openhole_2293 := [[458.14, -21.51, 181.39], [0.0395, 0.706003, 0.706809, -0.020511], [0,0,0,0], [9E9, 9E9, 9E9, 9E9, 9E9, 9E9]];
	VAR robtarget Openhole_2294 := [[458.64, -21.5, 181.4], [0.041123, 0.70591, 0.706756, -0.022258], [0,0,0,0], [9E9, 9E9, 9E9, 9E9, 9E9, 9E9]];
	VAR robtarget Openhole_2295 := [[459.14, -21.49, 181.41], [0.042797, 0.70581, 0.706701, -0.023953], [0,0,0,0], [9E9, 9E9, 9E9, 9E9, 9E9, 9E9]];
	VAR robtarget Openhole_2296 := [[459.64, -21.51, 181.43], [0.044513, 0.705704, 0.706643, -0.025602], [0,0,0,0], [9E9, 9E9, 9E9, 9E9, 9E9, 9E9]];
	VAR robtarget Openhole_2297 := [[460.14, -21.53, 181.44], [0.046272, 0.705591, 0.706583, -0.0272], [0,0,0,0], [9E9, 9E9, 9E9, 9E9, 9E9, 9E9]];
	VAR robtarget Openhole_2298 := [[461.64, -21.66, 181.49], [0.051687, 0.705215, 0.706391, -0.031806], [0,0,0,0], [9E9, 9E9, 9E9, 9E9, 9E9, 9E9]];
	VAR robtarget Openhole_2299 := [[467.1, -22.22, 181.73], [0.07158, 0.703474, 0.70546, -0.048231], [0,0,0,0], [9E9, 9E9, 9E9, 9E9, 9E9, 9E9]];
	VAR robtarget Openhole_2300 := [[475.59, -22.52, 182.06], [0.099742, 0.700037, 0.703118, -0.074998], [0,0,0,0], [9E9, 9E9, 9E9, 9E9, 9E9, 9E9]];
	VAR robtarget Openhole_2301 := [[485.58, -22.61, 182.43], [0.130391, 0.694981, 0.699117, -0.105994], [0,0,0,0], [9E9, 9E9, 9E9, 9E9, 9E9, 9E9]];
	VAR robtarget Openhole_2302 := [[486.08, -22.61, 182.45], [0.131854, 0.694705, 0.698885, -0.107514], [0,0,0,0], [9E9, 9E9, 9E9, 9E9, 9E9, 9E9]];
	VAR robtarget Openhole_2303 := [[497.58, -22.45, 182.77], [0.163571, 0.687928, 0.692802, -0.14151], [0,0,0,0], [9E9, 9E9, 9E9, 9E9, 9E9, 9E9]];
	VAR robtarget Openhole_2304 := [[504.35, -22.17, 182.84], [0.180364, 0.683717, 0.688601, -0.160713], [0,0,0,0], [9E9, 9E9, 9E9, 9E9, 9E9, 9E9]];
	VAR robtarget Openhole_2305 := [[509.35, -22.17, 183], [0.183051, 0.683002, 0.683002, -0.183051], [0,0,0,0], [9E9, 9E9, 9E9, 9E9, 9E9, 9E9]];
	VAR robtarget Openhole_2306 := [[536.35, -22.17, 182.91], [0.183051, 0.683002, 0.683002, -0.183051], [0,0,0,0], [9E9, 9E9, 9E9, 9E9, 9E9, 9E9]];
	VAR robtarget Openhole_2307 := [[536.35, -20.6, 182], [0.183051, 0.683002, 0.683002, -0.183051], [0,0,0,0], [9E9, 9E9, 9E9, 9E9, 9E9, 9E9]];
	VAR robtarget Openhole_2308 := [[509.35, -20.6, 182.09], [0.183051, 0.683002, 0.683002, -0.183051], [0,0,0,0], [9E9, 9E9, 9E9, 9E9, 9E9, 9E9]];
	VAR robtarget Openhole_2309 := [[504.35, -20.6, 182.01], [0.17579, 0.684907, 0.687511, -0.165314], [0,0,0,0], [9E9, 9E9, 9E9, 9E9, 9E9, 9E9]];
	VAR robtarget Openhole_2310 := [[495.11, -20.93, 182.02], [0.152298, 0.690511, 0.693268, -0.139211], [0,0,0,0], [9E9, 9E9, 9E9, 9E9, 9E9, 9E9]];
	VAR robtarget Openhole_2311 := [[489.11, -20.98, 181.93], [0.135566, 0.69399, 0.696554, -0.121707], [0,0,0,0], [9E9, 9E9, 9E9, 9E9, 9E9, 9E9]];
	VAR robtarget Openhole_2312 := [[488.61, -20.98, 181.92], [0.134121, 0.694271, 0.69681, -0.12023], [0,0,0,0], [9E9, 9E9, 9E9, 9E9, 9E9, 9E9]];
	VAR robtarget Openhole_2313 := [[474.12, -20.75, 181.59], [0.089332, 0.701441, 0.703004, -0.076061], [0,0,0,0], [9E9, 9E9, 9E9, 9E9, 9E9, 9E9]];
	VAR robtarget Openhole_2314 := [[464.13, -20.42, 181.38], [0.055803, 0.704901, 0.705716, -0.044321], [0,0,0,0], [9E9, 9E9, 9E9, 9E9, 9E9, 9E9]];
	VAR robtarget Openhole_2315 := [[462.63, -20.37, 181.35], [0.050628, 0.705292, 0.706002, -0.039505], [0,0,0,0], [9E9, 9E9, 9E9, 9E9, 9E9, 9E9]];
	VAR robtarget Openhole_2316 := [[461.63, -20.35, 181.34], [0.047242, 0.705527, 0.706179, -0.036203], [0,0,0,0], [9E9, 9E9, 9E9, 9E9, 9E9, 9E9]];
	VAR robtarget Openhole_2317 := [[460.13, -20.37, 181.32], [0.042304, 0.70584, 0.706424, -0.031075], [0,0,0,0], [9E9, 9E9, 9E9, 9E9, 9E9, 9E9]];
	VAR robtarget Openhole_2318 := [[459.13, -20.43, 181.31], [0.039143, 0.706023, 0.706571, -0.027516], [0,0,0,0], [9E9, 9E9, 9E9, 9E9, 9E9, 9E9]];
	VAR robtarget Openhole_2319 := [[458.63, -20.47, 181.31], [0.037606, 0.706106, 0.70664, -0.025693], [0,0,0,0], [9E9, 9E9, 9E9, 9E9, 9E9, 9E9]];
	VAR robtarget Openhole_2320 := [[457.64, -20.63, 181.31], [0.034844, 0.706248, 0.706771, -0.021796], [0,0,0,0], [9E9, 9E9, 9E9, 9E9, 9E9, 9E9]];
	VAR robtarget Openhole_2321 := [[457.1, -20.66, 181.3], [0.033111, 0.706331, 0.706828, -0.019865], [0,0,0,0], [9E9, 9E9, 9E9, 9E9, 9E9, 9E9]];
	VAR robtarget Openhole_2322 := [[454.66, -20.66, 181.26], [0.024842, 0.70667, 0.707012, -0.011555], [0,0,0,0], [9E9, 9E9, 9E9, 9E9, 9E9, 9E9]];
	VAR robtarget Openhole_2323 := [[454.85, -19.61, 181.21], [0.021929, 0.706767, 0.706931, -0.015776], [0,0,0,0], [9E9, 9E9, 9E9, 9E9, 9E9, 9E9]];
	VAR robtarget Openhole_2324 := [[457.29, -19.61, 181.23], [0.030202, 0.706461, 0.706697, -0.024078], [0,0,0,0], [9E9, 9E9, 9E9, 9E9, 9E9, 9E9]];
	VAR robtarget Openhole_2325 := [[458.04, -19.56, 181.23], [0.032529, 0.706358, 0.7066, -0.02676], [0,0,0,0], [9E9, 9E9, 9E9, 9E9, 9E9, 9E9]];
	VAR robtarget Openhole_2326 := [[460.01, -19.25, 181.2], [0.038126, 0.706078, 0.706266, -0.034479], [0,0,0,0], [9E9, 9E9, 9E9, 9E9, 9E9, 9E9]];
	VAR robtarget Openhole_2327 := [[463.43, -18.53, 181.11], [0.047143, 0.705534, 0.705449, -0.048395], [0,0,0,0], [9E9, 9E9, 9E9, 9E9, 9E9, 9E9]];
	VAR robtarget Openhole_2328 := [[464.4, -18.28, 181.07], [0.049542, 0.705369, 0.705159, -0.052446], [0,0,0,0], [9E9, 9E9, 9E9, 9E9, 9E9, 9E9]];
	VAR robtarget Openhole_2329 := [[465.37, -18.02, 181.03], [0.051839, 0.705204, 0.704843, -0.056539], [0,0,0,0], [9E9, 9E9, 9E9, 9E9, 9E9, 9E9]];
	VAR robtarget Openhole_2330 := [[467.31, -17.54, 180.92], [0.056662, 0.704833, 0.704156, -0.064536], [0,0,0,0], [9E9, 9E9, 9E9, 9E9, 9E9, 9E9]];
	VAR robtarget Openhole_2331 := [[467.8, -17.44, 180.9], [0.05794, 0.704729, 0.703975, -0.066477], [0,0,0,0], [9E9, 9E9, 9E9, 9E9, 9E9, 9E9]];
	VAR robtarget Openhole_2332 := [[468.29, -17.35, 180.88], [0.059257, 0.704619, 0.703792, -0.068386], [0,0,0,0], [9E9, 9E9, 9E9, 9E9, 9E9, 9E9]];
	VAR robtarget Openhole_2333 := [[470.26, -17.06, 180.79], [0.064759, 0.704135, 0.703032, -0.075799], [0,0,0,0], [9E9, 9E9, 9E9, 9E9, 9E9, 9E9]];
	VAR robtarget Openhole_2334 := [[471.26, -16.95, 180.74], [0.067627, 0.703865, 0.702637, -0.07938], [0,0,0,0], [9E9, 9E9, 9E9, 9E9, 9E9, 9E9]];
	VAR robtarget Openhole_2335 := [[476.25, -16.75, 180.59], [0.082993, 0.702219, 0.700561, -0.095988], [0,0,0,0], [9E9, 9E9, 9E9, 9E9, 9E9, 9E9]];
	VAR robtarget Openhole_2336 := [[478.25, -16.73, 180.54], [0.089265, 0.70145, 0.699668, -0.102296], [0,0,0,0], [9E9, 9E9, 9E9, 9E9, 9E9, 9E9]];
	VAR robtarget Openhole_2337 := [[478.75, -16.74, 180.53], [0.090837, 0.701248, 0.699439, -0.103848], [0,0,0,0], [9E9, 9E9, 9E9, 9E9, 9E9, 9E9]];
	VAR robtarget Openhole_2338 := [[491.74, -16.89, 180.31], [0.130448, 0.69497, 0.692684, -0.142088], [0,0,0,0], [9E9, 9E9, 9E9, 9E9, 9E9, 9E9]];
	VAR robtarget Openhole_2339 := [[492.24, -16.89, 180.3], [0.131882, 0.694699, 0.692391, -0.143509], [0,0,0,0], [9E9, 9E9, 9E9, 9E9, 9E9, 9E9]];
	VAR robtarget Openhole_2340 := [[500.74, -16.7, 180.03], [0.15491, 0.68993, 0.687029, -0.167306], [0,0,0,0], [9E9, 9E9, 9E9, 9E9, 9E9, 9E9]];
	VAR robtarget Openhole_2341 := [[504.34, -16.49, 179.84], [0.163823, 0.687868, 0.684524, -0.177278], [0,0,0,0], [9E9, 9E9, 9E9, 9E9, 9E9, 9E9]];
	VAR robtarget Openhole_2342 := [[509.34, -16.49, 179.72], [0.183051, 0.683002, 0.683002, -0.183051], [0,0,0,0], [9E9, 9E9, 9E9, 9E9, 9E9, 9E9]];
	VAR robtarget Openhole_2343 := [[536.34, -16.49, 179.63], [0.183051, 0.683002, 0.683002, -0.183051], [0,0,0,0], [9E9, 9E9, 9E9, 9E9, 9E9, 9E9]];
	VAR robtarget Openhole_2344 := [[536.33, -12.58, 177.38], [0.183051, 0.683002, 0.683002, -0.183051], [0,0,0,0], [9E9, 9E9, 9E9, 9E9, 9E9, 9E9]];
	VAR robtarget Openhole_2345 := [[509.33, -12.58, 177.46], [0.183051, 0.683002, 0.683002, -0.183051], [0,0,0,0], [9E9, 9E9, 9E9, 9E9, 9E9, 9E9]];
	VAR robtarget Openhole_2346 := [[504.34, -12.58, 177.77], [0.152383, 0.690492, 0.681486, -0.188617], [0,0,0,0], [9E9, 9E9, 9E9, 9E9, 9E9, 9E9]];
	VAR robtarget Openhole_2347 := [[498.82, -12.86, 178.24], [0.138198, 0.693471, 0.685447, -0.173674], [0,0,0,0], [9E9, 9E9, 9E9, 9E9, 9E9, 9E9]];
	VAR robtarget Openhole_2348 := [[495.33, -12.89, 178.47], [0.128459, 0.69534, 0.687766, -0.16425], [0,0,0,0], [9E9, 9E9, 9E9, 9E9, 9E9, 9E9]];
	VAR robtarget Openhole_2349 := [[494.83, -12.89, 178.49], [0.127024, 0.695604, 0.688087, -0.162901], [0,0,0,0], [9E9, 9E9, 9E9, 9E9, 9E9, 9E9]];
	VAR robtarget Openhole_2350 := [[482.35, -12.7, 179.17], [0.089088, 0.701472, 0.695464, -0.127791], [0,0,0,0], [9E9, 9E9, 9E9, 9E9, 9E9, 9E9]];
	VAR robtarget Openhole_2351 := [[481.85, -12.7, 179.2], [0.087538, 0.701667, 0.695738, -0.126288], [0,0,0,0], [9E9, 9E9, 9E9, 9E9, 9E9, 9E9]];
	VAR robtarget Openhole_2352 := [[476.37, -12.88, 179.58], [0.070727, 0.703561, 0.69866, -0.108972], [0,0,0,0], [9E9, 9E9, 9E9, 9E9, 9E9, 9E9]];
	VAR robtarget Openhole_2353 := [[472.41, -13.34, 179.92], [0.059438, 0.704604, 0.700696, -0.095002], [0,0,0,0], [9E9, 9E9, 9E9, 9E9, 9E9, 9E9]];
	VAR robtarget Openhole_2354 := [[471.92, -13.42, 179.96], [0.058103, 0.704716, 0.700942, -0.093168], [0,0,0,0], [9E9, 9E9, 9E9, 9E9, 9E9, 9E9]];
	VAR robtarget Openhole_2355 := [[470.94, -13.62, 180.06], [0.05556, 0.704921, 0.701433, -0.089395], [0,0,0,0], [9E9, 9E9, 9E9, 9E9, 9E9, 9E9]];
	VAR robtarget Openhole_2356 := [[470.46, -13.73, 180.1], [0.054332, 0.705016, 0.701676, -0.087473], [0,0,0,0], [9E9, 9E9, 9E9, 9E9, 9E9, 9E9]];
	VAR robtarget Openhole_2357 := [[469.49, -13.97, 180.2], [0.051958, 0.705195, 0.702152, -0.083558], [0,0,0,0], [9E9, 9E9, 9E9, 9E9, 9E9, 9E9]];
	VAR robtarget Openhole_2358 := [[468.53, -14.24, 180.3], [0.049697, 0.705358, 0.702617, -0.079556], [0,0,0,0], [9E9, 9E9, 9E9, 9E9, 9E9, 9E9]];
	VAR robtarget Openhole_2359 := [[467.59, -14.54, 180.39], [0.047582, 0.705504, 0.703069, -0.075455], [0,0,0,0], [9E9, 9E9, 9E9, 9E9, 9E9, 9E9]];
	VAR robtarget Openhole_2360 := [[467.12, -14.71, 180.44], [0.046585, 0.705571, 0.70329, -0.073367], [0,0,0,0], [9E9, 9E9, 9E9, 9E9, 9E9, 9E9]];
	VAR robtarget Openhole_2361 := [[466.65, -14.89, 180.49], [0.045636, 0.705633, 0.703508, -0.071252], [0,0,0,0], [9E9, 9E9, 9E9, 9E9, 9E9, 9E9]];
	VAR robtarget Openhole_2362 := [[466.19, -15.08, 180.54], [0.04474, 0.70569, 0.703721, -0.069109], [0,0,0,0], [9E9, 9E9, 9E9, 9E9, 9E9, 9E9]];
	VAR robtarget Openhole_2363 := [[465.73, -15.28, 180.59], [0.043885, 0.705744, 0.703931, -0.066945], [0,0,0,0], [9E9, 9E9, 9E9, 9E9, 9E9, 9E9]];
	VAR robtarget Openhole_2364 := [[464.83, -15.7, 180.69], [0.042291, 0.705841, 0.704334, -0.062559], [0,0,0,0], [9E9, 9E9, 9E9, 9E9, 9E9, 9E9]];
	VAR robtarget Openhole_2365 := [[463.94, -16.14, 180.78], [0.040824, 0.705927, 0.704715, -0.05811], [0,0,0,0], [9E9, 9E9, 9E9, 9E9, 9E9, 9E9]];
	VAR robtarget Openhole_2366 := [[462.19, -17.09, 180.94], [0.038131, 0.706078, 0.705401, -0.049086], [0,0,0,0], [9E9, 9E9, 9E9, 9E9, 9E9, 9E9]];
	VAR robtarget Openhole_2367 := [[461.3, -17.54, 181.01], [0.036696, 0.706154, 0.7057, -0.044578], [0,0,0,0], [9E9, 9E9, 9E9, 9E9, 9E9, 9E9]];
	VAR robtarget Openhole_2368 := [[460.84, -17.74, 181.04], [0.035801, 0.7062, 0.705835, -0.042382], [0,0,0,0], [9E9, 9E9, 9E9, 9E9, 9E9, 9E9]];
	VAR robtarget Openhole_2369 := [[460.37, -17.92, 181.06], [0.034851, 0.706247, 0.705963, -0.040206], [0,0,0,0], [9E9, 9E9, 9E9, 9E9, 9E9, 9E9]];
	VAR robtarget Openhole_2370 := [[459.42, -18.22, 181.1], [0.032652, 0.706353, 0.70619, -0.035989], [0,0,0,0], [9E9, 9E9, 9E9, 9E9, 9E9, 9E9]];
	VAR robtarget Openhole_2371 := [[458.45, -18.46, 181.13], [0.030212, 0.706461, 0.706387, -0.031893], [0,0,0,0], [9E9, 9E9, 9E9, 9E9, 9E9, 9E9]];
	VAR robtarget Openhole_2372 := [[457.96, -18.57, 181.14], [0.028935, 0.706515, 0.706475, -0.029876], [0,0,0,0], [9E9, 9E9, 9E9, 9E9, 9E9, 9E9]];
	VAR robtarget Openhole_2373 := [[457.34, -18.58, 181.15], [0.026868, 0.706596, 0.706562, -0.027763], [0,0,0,0], [9E9, 9E9, 9E9, 9E9, 9E9, 9E9]];
	VAR robtarget Openhole_2374 := [[454.9, -18.58, 181.16], [0.018589, 0.706862, 0.706839, -0.019468], [0,0,0,0], [9E9, 9E9, 9E9, 9E9, 9E9, 9E9]];
	VAR robtarget Openhole_2375 := [[454.82, -17.6, 181.11], [0.015016, 0.706947, 0.706748, -0.022534], [0,0,0,0], [9E9, 9E9, 9E9, 9E9, 9E9, 9E9]];
	VAR robtarget Openhole_2376 := [[457.27, -17.6, 181.07], [0.023302, 0.706723, 0.706435, -0.030823], [0,0,0,0], [9E9, 9E9, 9E9, 9E9, 9E9, 9E9]];
	VAR robtarget Openhole_2377 := [[457.88, -17.43, 181.05], [0.024808, 0.706671, 0.706315, -0.03346], [0,0,0,0], [9E9, 9E9, 9E9, 9E9, 9E9, 9E9]];
	VAR robtarget Openhole_2378 := [[458.35, -17.26, 181.03], [0.025819, 0.706635, 0.706209, -0.035621], [0,0,0,0], [9E9, 9E9, 9E9, 9E9, 9E9, 9E9]];
	VAR robtarget Openhole_2379 := [[458.82, -17.08, 181], [0.026773, 0.7066, 0.706095, -0.037805], [0,0,0,0], [9E9, 9E9, 9E9, 9E9, 9E9, 9E9]];
	VAR robtarget Openhole_2380 := [[459.27, -16.88, 180.98], [0.02762, 0.706567, 0.705973, -0.040029], [0,0,0,0], [9E9, 9E9, 9E9, 9E9, 9E9, 9E9]];
	VAR robtarget Openhole_2381 := [[459.72, -16.65, 180.94], [0.028375, 0.706537, 0.705841, -0.042283], [0,0,0,0], [9E9, 9E9, 9E9, 9E9, 9E9, 9E9]];
	VAR robtarget Openhole_2382 := [[460.15, -16.4, 180.91], [0.028968, 0.706513, 0.7057, -0.044582], [0,0,0,0], [9E9, 9E9, 9E9, 9E9, 9E9, 9E9]];
	VAR robtarget Openhole_2383 := [[461.82, -15.31, 180.74], [0.030923, 0.70643, 0.705054, -0.053836], [0,0,0,0], [9E9, 9E9, 9E9, 9E9, 9E9, 9E9]];
	VAR robtarget Openhole_2384 := [[463.11, -14.56, 180.59], [0.032729, 0.706349, 0.704501, -0.060655], [0,0,0,0], [9E9, 9E9, 9E9, 9E9, 9E9, 9E9]];
	VAR robtarget Openhole_2385 := [[464.88, -13.66, 180.38], [0.035621, 0.706209, 0.703679, -0.069544], [0,0,0,0], [9E9, 9E9, 9E9, 9E9, 9E9, 9E9]];
	VAR robtarget Openhole_2386 := [[465.33, -13.45, 180.32], [0.036442, 0.706167, 0.70346, -0.07172], [0,0,0,0], [9E9, 9E9, 9E9, 9E9, 9E9, 9E9]];
	VAR robtarget Openhole_2387 := [[465.79, -13.26, 180.27], [0.037321, 0.706121, 0.703238, -0.07387], [0,0,0,0], [9E9, 9E9, 9E9, 9E9, 9E9, 9E9]];
	VAR robtarget Openhole_2388 := [[466.25, -13.07, 180.21], [0.038245, 0.706072, 0.703011, -0.075996], [0,0,0,0], [9E9, 9E9, 9E9, 9E9, 9E9, 9E9]];
	VAR robtarget Openhole_2389 := [[467.66, -12.58, 180.04], [0.041265, 0.705902, 0.702309, -0.082231], [0,0,0,0], [9E9, 9E9, 9E9, 9E9, 9E9, 9E9]];
	VAR robtarget Openhole_2390 := [[468.61, -12.29, 179.93], [0.043452, 0.70577, 0.701824, -0.086276], [0,0,0,0], [9E9, 9E9, 9E9, 9E9, 9E9, 9E9]];
	VAR robtarget Openhole_2391 := [[469.57, -12.03, 179.82], [0.045764, 0.705624, 0.701326, -0.090229], [0,0,0,0], [9E9, 9E9, 9E9, 9E9, 9E9, 9E9]];
	VAR robtarget Openhole_2392 := [[470.53, -11.8, 179.71], [0.048201, 0.705462, 0.70082, -0.094085], [0,0,0,0], [9E9, 9E9, 9E9, 9E9, 9E9, 9E9]];
	VAR robtarget Openhole_2393 := [[471.02, -11.7, 179.65], [0.049466, 0.705374, 0.700563, -0.095976], [0,0,0,0], [9E9, 9E9, 9E9, 9E9, 9E9, 9E9]];
	VAR robtarget Openhole_2394 := [[474.95, -11.1, 179.23], [0.06037, 0.704525, 0.698447, -0.110326], [0,0,0,0], [9E9, 9E9, 9E9, 9E9, 9E9, 9E9]];
	VAR robtarget Openhole_2395 := [[478.92, -10.84, 178.85], [0.072315, 0.703399, 0.696256, -0.123399], [0,0,0,0], [9E9, 9E9, 9E9, 9E9, 9E9, 9E9]];
	VAR robtarget Openhole_2396 := [[482.41, -10.79, 178.56], [0.083178, 0.702198, 0.694286, -0.134043], [0,0,0,0], [9E9, 9E9, 9E9, 9E9, 9E9, 9E9]];
	VAR robtarget Openhole_2397 := [[482.91, -10.8, 178.52], [0.084745, 0.70201, 0.694, -0.135513], [0,0,0,0], [9E9, 9E9, 9E9, 9E9, 9E9, 9E9]];
	VAR robtarget Openhole_2398 := [[497.37, -11.14, 177.54], [0.128968, 0.695246, 0.685117, -0.174971], [0,0,0,0], [9E9, 9E9, 9E9, 9E9, 9E9, 9E9]];
	VAR robtarget Openhole_2399 := [[497.87, -11.14, 177.5], [0.130376, 0.694984, 0.684779, -0.176287], [0,0,0,0], [9E9, 9E9, 9E9, 9E9, 9E9, 9E9]];
	VAR robtarget Openhole_2400 := [[502.85, -10.99, 177.04], [0.143689, 0.692354, 0.681234, -0.189525], [0,0,0,0], [9E9, 9E9, 9E9, 9E9, 9E9, 9E9]];
	VAR robtarget Openhole_2401 := [[504.39, -10.89, 176.87], [0.147578, 0.691535, 0.68007, -0.19366], [0,0,0,0], [9E9, 9E9, 9E9, 9E9, 9E9, 9E9]];
	VAR robtarget Openhole_2402 := [[509.33, -10.89, 176.48], [0.183051, 0.683002, 0.683002, -0.183051], [0,0,0,0], [9E9, 9E9, 9E9, 9E9, 9E9, 9E9]];
	VAR robtarget Openhole_2403 := [[536.33, -10.89, 176.4], [0.183051, 0.683002, 0.683002, -0.183051], [0,0,0,0], [9E9, 9E9, 9E9, 9E9, 9E9, 9E9]];
	VAR robtarget Openhole_2404 := [[536.33, -10, 175.89], [0.183051, 0.683002, 0.683002, -0.183051], [0,0,0,0], [9E9, 9E9, 9E9, 9E9, 9E9, 9E9]];
	VAR robtarget Openhole_2405 := [[509.33, -10, 175.97], [0.183051, 0.683002, 0.683002, -0.183051], [0,0,0,0], [9E9, 9E9, 9E9, 9E9, 9E9, 9E9]];
	VAR robtarget Openhole_2406 := [[504.33, -10, 176.41], [0.144832, 0.692115, 0.679385, -0.196051], [0,0,0,0], [9E9, 9E9, 9E9, 9E9, 9E9, 9E9]];
	VAR robtarget Openhole_2407 := [[503.56, -10.02, 176.48], [0.142771, 0.692543, 0.679946, -0.194097], [0,0,0,0], [9E9, 9E9, 9E9, 9E9, 9E9, 9E9]];
	VAR robtarget Openhole_2408 := [[499.58, -10.13, 176.88], [0.132127, 0.694653, 0.682819, -0.183733], [0,0,0,0], [9E9, 9E9, 9E9, 9E9, 9E9, 9E9]];
	VAR robtarget Openhole_2409 := [[499.08, -10.12, 176.92], [0.130723, 0.694918, 0.683162, -0.182454], [0,0,0,0], [9E9, 9E9, 9E9, 9E9, 9E9, 9E9]];
	VAR robtarget Openhole_2410 := [[490.61, -9.87, 177.54], [0.10537, 0.699212, 0.688654, -0.160487], [0,0,0,0], [9E9, 9E9, 9E9, 9E9, 9E9, 9E9]];
	VAR robtarget Openhole_2411 := [[482.14, -9.61, 178.21], [0.078542, 0.702731, 0.693715, -0.136967], [0,0,0,0], [9E9, 9E9, 9E9, 9E9, 9E9, 9E9]];
	VAR robtarget Openhole_2412 := [[481.64, -9.62, 178.26], [0.076976, 0.702904, 0.694006, -0.135486], [0,0,0,0], [9E9, 9E9, 9E9, 9E9, 9E9, 9E9]];
	VAR robtarget Openhole_2413 := [[476.67, -9.77, 178.75], [0.061587, 0.70442, 0.696859, -0.119948], [0,0,0,0], [9E9, 9E9, 9E9, 9E9, 9E9, 9E9]];
	VAR robtarget Openhole_2414 := [[472.72, -10.2, 179.2], [0.050124, 0.705328, 0.699078, -0.106251], [0,0,0,0], [9E9, 9E9, 9E9, 9E9, 9E9, 9E9]];
	VAR robtarget Openhole_2415 := [[469.79, -10.75, 179.55], [0.042289, 0.705841, 0.700676, -0.095145], [0,0,0,0], [9E9, 9E9, 9E9, 9E9, 9E9, 9E9]];
	VAR robtarget Openhole_2416 := [[466.45, -11.71, 179.98], [0.034356, 0.706272, 0.70243, -0.081189], [0,0,0,0], [9E9, 9E9, 9E9, 9E9, 9E9, 9E9]];
	VAR robtarget Openhole_2417 := [[465.51, -12.04, 180.09], [0.032326, 0.706367, 0.702899, -0.07703], [0,0,0,0], [9E9, 9E9, 9E9, 9E9, 9E9, 9E9]];
	VAR robtarget Openhole_2418 := [[465.05, -12.22, 180.15], [0.031383, 0.70641, 0.703128, -0.074911], [0,0,0,0], [9E9, 9E9, 9E9, 9E9, 9E9, 9E9]];
	VAR robtarget Openhole_2419 := [[463.68, -12.81, 180.32], [0.028764, 0.706521, 0.703787, -0.068436], [0,0,0,0], [9E9, 9E9, 9E9, 9E9, 9E9, 9E9]];
	VAR robtarget Openhole_2420 := [[463.23, -13.02, 180.38], [0.027963, 0.706554, 0.703997, -0.066241], [0,0,0,0], [9E9, 9E9, 9E9, 9E9, 9E9, 9E9]];
	VAR robtarget Openhole_2421 := [[461.03, -14.18, 180.64], [0.024466, 0.706683, 0.704962, -0.055032], [0,0,0,0], [9E9, 9E9, 9E9, 9E9, 9E9, 9E9]];
	VAR robtarget Openhole_2422 := [[460.18, -14.69, 180.73], [0.023293, 0.706723, 0.705304, -0.050456], [0,0,0,0], [9E9, 9E9, 9E9, 9E9, 9E9, 9E9]];
	VAR robtarget Openhole_2423 := [[459.34, -15.23, 180.82], [0.022292, 0.706755, 0.70562, -0.045825], [0,0,0,0], [9E9, 9E9, 9E9, 9E9, 9E9, 9E9]];
	VAR robtarget Openhole_2424 := [[458.92, -15.49, 180.86], [0.02174, 0.706772, 0.705766, -0.043517], [0,0,0,0], [9E9, 9E9, 9E9, 9E9, 9E9, 9E9]];
	VAR robtarget Openhole_2425 := [[458.48, -15.74, 180.89], [0.021115, 0.706791, 0.705904, -0.041222], [0,0,0,0], [9E9, 9E9, 9E9, 9E9, 9E9, 9E9]];
	VAR robtarget Openhole_2426 := [[457.6, -16.2, 180.96], [0.019674, 0.706833, 0.706155, -0.03668], [0,0,0,0], [9E9, 9E9, 9E9, 9E9, 9E9, 9E9]];
	VAR robtarget Openhole_2427 := [[457.02, -16.45, 180.99], [0.018588, 0.706862, 0.706295, -0.033878], [0,0,0,0], [9E9, 9E9, 9E9, 9E9, 9E9, 9E9]];
	VAR robtarget Openhole_2428 := [[454.58, -16.45, 181.05], [0.010292, 0.707032, 0.706643, -0.025593], [0,0,0,0], [9E9, 9E9, 9E9, 9E9, 9E9, 9E9]];
	VAR robtarget Openhole_2429 := [[454.01, -15.03, 181], [0.003534, 0.707098, 0.706533, -0.02849], [0,0,0,0], [9E9, 9E9, 9E9, 9E9, 9E9, 9E9]];
	VAR robtarget Openhole_2430 := [[456.45, -15.03, 180.91], [0.011842, 0.707008, 0.70615, -0.036773], [0,0,0,0], [9E9, 9E9, 9E9, 9E9, 9E9, 9E9]];
	VAR robtarget Openhole_2431 := [[457.91, -14.13, 180.78], [0.013707, 0.706974, 0.70569, -0.044737], [0,0,0,0], [9E9, 9E9, 9E9, 9E9, 9E9, 9E9]];
	VAR robtarget Openhole_2432 := [[458.76, -13.61, 180.69], [0.01486, 0.706951, 0.705383, -0.049341], [0,0,0,0], [9E9, 9E9, 9E9, 9E9, 9E9, 9E9]];
	VAR robtarget Openhole_2433 := [[459.2, -13.37, 180.65], [0.015537, 0.706936, 0.705221, -0.051611], [0,0,0,0], [9E9, 9E9, 9E9, 9E9, 9E9, 9E9]];
	VAR robtarget Openhole_2434 := [[459.64, -13.14, 180.6], [0.016258, 0.70692, 0.705052, -0.053864], [0,0,0,0], [9E9, 9E9, 9E9, 9E9, 9E9, 9E9]];
	VAR robtarget Openhole_2435 := [[460.53, -12.71, 180.5], [0.017819, 0.706882, 0.704698, -0.058319], [0,0,0,0], [9E9, 9E9, 9E9, 9E9, 9E9, 9E9]];
	VAR robtarget Openhole_2436 := [[461.9, -12.1, 180.34], [0.020385, 0.706813, 0.704123, -0.064891], [0,0,0,0], [9E9, 9E9, 9E9, 9E9, 9E9, 9E9]];
	VAR robtarget Openhole_2437 := [[463.74, -11.36, 180.12], [0.024122, 0.706695, 0.70328, -0.073463], [0,0,0,0], [9E9, 9E9, 9E9, 9E9, 9E9, 9E9]];
	VAR robtarget Openhole_2438 := [[466.57, -10.43, 179.76], [0.030468, 0.70645, 0.701878, -0.085833], [0,0,0,0], [9E9, 9E9, 9E9, 9E9, 9E9, 9E9]];
	VAR robtarget Openhole_2439 := [[468.97, -9.8, 179.44], [0.036394, 0.70617, 0.700607, -0.095653], [0,0,0,0], [9E9, 9E9, 9E9, 9E9, 9E9, 9E9]];
	VAR robtarget Openhole_2440 := [[472.87, -9.09, 178.93], [0.04696, 0.705546, 0.69844, -0.11037], [0,0,0,0], [9E9, 9E9, 9E9, 9E9, 9E9, 9E9]];
	VAR robtarget Openhole_2441 := [[477.32, -8.67, 178.39], [0.060095, 0.704548, 0.695882, -0.125493], [0,0,0,0], [9E9, 9E9, 9E9, 9E9, 9E9, 9E9]];
	VAR robtarget Openhole_2442 := [[481.79, -8.56, 177.91], [0.074075, 0.703216, 0.693257, -0.139265], [0,0,0,0], [9E9, 9E9, 9E9, 9E9, 9E9, 9E9]];
	VAR robtarget Openhole_2443 := [[482.29, -8.56, 177.86], [0.075653, 0.703048, 0.692961, -0.14073], [0,0,0,0], [9E9, 9E9, 9E9, 9E9, 9E9, 9E9]];
	VAR robtarget Openhole_2444 := [[490.75, -8.89, 177.14], [0.102747, 0.699602, 0.687852, -0.163888], [0,0,0,0], [9E9, 9E9, 9E9, 9E9, 9E9, 9E9]];
	VAR robtarget Openhole_2445 := [[499.21, -9.25, 176.49], [0.1285, 0.695333, 0.682376, -0.185371], [0,0,0,0], [9E9, 9E9, 9E9, 9E9, 9E9, 9E9]];
	VAR robtarget Openhole_2446 := [[500.21, -9.26, 176.4], [0.131319, 0.694806, 0.681685, -0.187897], [0,0,0,0], [9E9, 9E9, 9E9, 9E9, 9E9, 9E9]];
	VAR robtarget Openhole_2447 := [[500.71, -9.26, 176.35], [0.132697, 0.694544, 0.681333, -0.189172], [0,0,0,0], [9E9, 9E9, 9E9, 9E9, 9E9, 9E9]];
	VAR robtarget Openhole_2448 := [[503.19, -9.2, 176.09], [0.139402, 0.693229, 0.67953, -0.195549], [0,0,0,0], [9E9, 9E9, 9E9, 9E9, 9E9, 9E9]];
	VAR robtarget Openhole_2449 := [[503.69, -9.17, 176.03], [0.140657, 0.692976, 0.67915, -0.196864], [0,0,0,0], [9E9, 9E9, 9E9, 9E9, 9E9, 9E9]];
	VAR robtarget Openhole_2450 := [[504.33, -9.15, 175.95], [0.14232, 0.692636, 0.678669, -0.198515], [0,0,0,0], [9E9, 9E9, 9E9, 9E9, 9E9, 9E9]];
	VAR robtarget Openhole_2451 := [[509.33, -9.15, 175.48], [0.183051, 0.683002, 0.683002, -0.183051], [0,0,0,0], [9E9, 9E9, 9E9, 9E9, 9E9, 9E9]];
	VAR robtarget Openhole_2452 := [[536.33, -9.15, 175.39], [0.183051, 0.683002, 0.683002, -0.183051], [0,0,0,0], [9E9, 9E9, 9E9, 9E9, 9E9, 9E9]];
	VAR robtarget Openhole_2453 := [[536.33, -8.27, 174.89], [0.183051, 0.683002, 0.683002, -0.183051], [0,0,0,0], [9E9, 9E9, 9E9, 9E9, 9E9, 9E9]];
	VAR robtarget Openhole_2454 := [[524.33, -8.27, 174.93], [0.183051, 0.683002, 0.683002, -0.183051], [0,0,0,0], [9E9, 9E9, 9E9, 9E9, 9E9, 9E9]];
	VAR robtarget Openhole_2455 := [[509.33, -8.28, 174.97], [0.183051, 0.683002, 0.683002, -0.183051], [0,0,0,0], [9E9, 9E9, 9E9, 9E9, 9E9, 9E9]];
	VAR robtarget Openhole_2456 := [[504.35, -8.28, 175.49], [0.139846, 0.69314, 0.677918, -0.201066], [0,0,0,0], [9E9, 9E9, 9E9, 9E9, 9E9, 9E9]];
	VAR robtarget Openhole_2457 := [[503.83, -8.3, 175.56], [0.138508, 0.693409, 0.678316, -0.199719], [0,0,0,0], [9E9, 9E9, 9E9, 9E9, 9E9, 9E9]];
	VAR robtarget Openhole_2458 := [[501.35, -8.33, 175.82], [0.131725, 0.694729, 0.680118, -0.193494], [0,0,0,0], [9E9, 9E9, 9E9, 9E9, 9E9, 9E9]];
	VAR robtarget Openhole_2459 := [[500.85, -8.32, 175.87], [0.13032, 0.694994, 0.680468, -0.19226], [0,0,0,0], [9E9, 9E9, 9E9, 9E9, 9E9, 9E9]];
	VAR robtarget Openhole_2460 := [[493.88, -7.98, 176.44], [0.109266, 0.698614, 0.685063, -0.17518], [0,0,0,0], [9E9, 9E9, 9E9, 9E9, 9E9, 9E9]];
	VAR robtarget Openhole_2461 := [[483.94, -7.4, 177.31], [0.077165, 0.702884, 0.691186, -0.149203], [0,0,0,0], [9E9, 9E9, 9E9, 9E9, 9E9, 9E9]];
	VAR robtarget Openhole_2462 := [[480.96, -7.35, 177.63], [0.067561, 0.703872, 0.692983, -0.14062], [0,0,0,0], [9E9, 9E9, 9E9, 9E9, 9E9, 9E9]];
	VAR robtarget Openhole_2463 := [[480.46, -7.35, 177.68], [0.065979, 0.704022, 0.693282, -0.139141], [0,0,0,0], [9E9, 9E9, 9E9, 9E9, 9E9, 9E9]];
	VAR robtarget Openhole_2464 := [[476, -7.51, 178.23], [0.052047, 0.705189, 0.695939, -0.125175], [0,0,0,0], [9E9, 9E9, 9E9, 9E9, 9E9, 9E9]];
	VAR robtarget Openhole_2465 := [[471.56, -7.98, 178.82], [0.039008, 0.70603, 0.698521, -0.109858], [0,0,0,0], [9E9, 9E9, 9E9, 9E9, 9E9, 9E9]];
	VAR robtarget Openhole_2466 := [[467.18, -8.8, 179.43], [0.027116, 0.706587, 0.70094, -0.093183], [0,0,0,0], [9E9, 9E9, 9E9, 9E9, 9E9, 9E9]];
	VAR robtarget Openhole_2467 := [[464.77, -9.39, 179.75], [0.020998, 0.706795, 0.702171, -0.083405], [0,0,0,0], [9E9, 9E9, 9E9, 9E9, 9E9, 9E9]];
	VAR robtarget Openhole_2468 := [[459.05, -11.07, 180.44], [0.007297, 0.707069, 0.704651, -0.058875], [0,0,0,0], [9E9, 9E9, 9E9, 9E9, 9E9, 9E9]];
	VAR robtarget Openhole_2469 := [[458.11, -11.38, 180.54], [0.005102, 0.707088, 0.704989, -0.054681], [0,0,0,0], [9E9, 9E9, 9E9, 9E9, 9E9, 9E9]];
	VAR robtarget Openhole_2470 := [[457.17, -11.7, 180.63], [0.003011, 0.7071, 0.705307, -0.050422], [0,0,0,0], [9E9, 9E9, 9E9, 9E9, 9E9, 9E9]];
	VAR robtarget Openhole_2471 := [[456.7, -11.89, 180.68], [0.002051, 0.707104, 0.705459, -0.048248], [0,0,0,0], [9E9, 9E9, 9E9, 9E9, 9E9, 9E9]];
	VAR robtarget Openhole_2472 := [[456.25, -12.09, 180.72], [0.0012, 0.707106, 0.705607, -0.046029], [0,0,0,0], [9E9, 9E9, 9E9, 9E9, 9E9, 9E9]];
	VAR robtarget Openhole_2473 := [[455.8, -12.3, 180.76], [0.000388, 0.707107, 0.70575, -0.043791], [0,0,0,0], [9E9, 9E9, 9E9, 9E9, 9E9, 9E9]];
	VAR robtarget Openhole_2474 := [[455.36, -12.53, 180.81], [-0.00035, 0.707107, 0.705886, -0.041525], [0,0,0,0], [9E9, 9E9, 9E9, 9E9, 9E9, 9E9]];
	VAR robtarget Openhole_2475 := [[454.82, -12.87, 180.86], [-0.001006, 0.707106, 0.706053, -0.038581], [0,0,0,0], [9E9, 9E9, 9E9, 9E9, 9E9, 9E9]];
	VAR robtarget Openhole_2476 := [[445.25, -11.83, 181.47], [-0.037068, 0.706135, 0.707042, -0.009578], [0,0,0,0], [9E9, 9E9, 9E9, 9E9, 9E9, 9E9]];
	VAR robtarget Openhole_2477 := [[444.72, -11.69, 181.51], [-0.039351, 0.706011, 0.707059, -0.008235], [0,0,0,0], [9E9, 9E9, 9E9, 9E9, 9E9, 9E9]];
	VAR robtarget Openhole_2478 := [[444.22, -11.62, 181.55], [-0.041235, 0.705903, 0.707074, -0.006763], [0,0,0,0], [9E9, 9E9, 9E9, 9E9, 9E9, 9E9]];
	VAR robtarget Openhole_2479 := [[443.23, -11.52, 181.62], [-0.044915, 0.705679, 0.707097, -0.003715], [0,0,0,0], [9E9, 9E9, 9E9, 9E9, 9E9, 9E9]];
	VAR robtarget Openhole_2480 := [[442.24, -11.45, 181.7], [-0.048507, 0.705441, 0.707107, -0.000573], [0,0,0,0], [9E9, 9E9, 9E9, 9E9, 9E9, 9E9]];
	VAR robtarget Openhole_2481 := [[441.74, -11.43, 181.74], [-0.050269, 0.705318, 0.707106, 0.001032], [0,0,0,0], [9E9, 9E9, 9E9, 9E9, 9E9, 9E9]];
	VAR robtarget Openhole_2482 := [[431.77, -11.25, 182.5], [-0.083838, 0.702119, 0.706282, 0.034138], [0,0,0,0], [9E9, 9E9, 9E9, 9E9, 9E9, 9E9]];
	VAR robtarget Openhole_2483 := [[431.27, -11.25, 182.53], [-0.085449, 0.701925, 0.706199, 0.03581], [0,0,0,0], [9E9, 9E9, 9E9, 9E9, 9E9, 9E9]];
	VAR robtarget Openhole_2484 := [[407.33, -11.81, 184.1], [-0.156227, 0.689633, 0.697943, 0.113472], [0,0,0,0], [9E9, 9E9, 9E9, 9E9, 9E9, 9E9]];
	VAR robtarget Openhole_2485 := [[396.35, -12.23, 184.65], [-0.184218, 0.682689, 0.691896, 0.145875], [0,0,0,0], [9E9, 9E9, 9E9, 9E9, 9E9, 9E9]];
	VAR robtarget Openhole_2486 := [[394.34, -12.34, 184.72], [-0.188963, 0.681391, 0.690659, 0.151623], [0,0,0,0], [9E9, 9E9, 9E9, 9E9, 9E9, 9E9]];
	VAR robtarget Openhole_2487 := [[389.36, -12.34, 185.04], [-0.201092, 0.67791, 0.687677, 0.164623], [0,0,0,0], [9E9, 9E9, 9E9, 9E9, 9E9, 9E9]];
	VAR robtarget Openhole_2488 := [[362.36, -12.34, 185.13], [-0.183051, 0.683002, 0.683002, 0.183051], [0,0,0,0], [9E9, 9E9, 9E9, 9E9, 9E9, 9E9]];
	VAR robtarget Openhole_2489 := [[362.36, -13.23, 184.62], [-0.183051, 0.683002, 0.683002, 0.183051], [0,0,0,0], [9E9, 9E9, 9E9, 9E9, 9E9, 9E9]];
	VAR robtarget Openhole_2490 := [[374.36, -13.23, 184.58], [-0.183051, 0.683002, 0.683002, 0.183051], [0,0,0,0], [9E9, 9E9, 9E9, 9E9, 9E9, 9E9]];
	VAR robtarget Openhole_2491 := [[389.36, -13.23, 184.53], [-0.198602, 0.678644, 0.687067, 0.167151], [0,0,0,0], [9E9, 9E9, 9E9, 9E9, 9E9, 9E9]];
	VAR robtarget Openhole_2492 := [[394.33, -13.23, 184.25], [-0.186414, 0.682092, 0.690084, 0.154219], [0,0,0,0], [9E9, 9E9, 9E9, 9E9, 9E9, 9E9]];
	VAR robtarget Openhole_2493 := [[404.34, -12.8, 183.88], [-0.161469, 0.688424, 0.695926, 0.125247], [0,0,0,0], [9E9, 9E9, 9E9, 9E9, 9E9, 9E9]];
	VAR robtarget Openhole_2494 := [[421.81, -12.49, 182.92], [-0.111428, 0.698272, 0.703543, 0.070905], [0,0,0,0], [9E9, 9E9, 9E9, 9E9, 9E9, 9E9]];
	VAR robtarget Openhole_2495 := [[427.8, -12.45, 182.54], [-0.092678, 0.701007, 0.705242, 0.051319], [0,0,0,0], [9E9, 9E9, 9E9, 9E9, 9E9, 9E9]];
	VAR robtarget Openhole_2496 := [[428.3, -12.46, 182.51], [-0.091074, 0.701217, 0.705359, 0.04968], [0,0,0,0], [9E9, 9E9, 9E9, 9E9, 9E9, 9E9]];
	VAR robtarget Openhole_2497 := [[434.78, -12.62, 182.08], [-0.069436, 0.703689, 0.706527, 0.028629], [0,0,0,0], [9E9, 9E9, 9E9, 9E9, 9E9, 9E9]];
	VAR robtarget Openhole_2498 := [[440.25, -13.05, 181.71], [-0.049813, 0.70535, 0.707012, 0.011575], [0,0,0,0], [9E9, 9E9, 9E9, 9E9, 9E9, 9E9]];
	VAR robtarget Openhole_2499 := [[442.74, -13.1, 181.56], [-0.041227, 0.705904, 0.707099, 0.003292], [0,0,0,0], [9E9, 9E9, 9E9, 9E9, 9E9, 9E9]];
	VAR robtarget Openhole_2500 := [[443.43, -13.31, 181.51], [-0.038198, 0.706074, 0.707105, 0.001644], [0,0,0,0], [9E9, 9E9, 9E9, 9E9, 9E9, 9E9]];
	VAR robtarget Openhole_2501 := [[445.21, -13.31, 181.41], [-0.032199, 0.706373, 0.707093, -0.004396], [0,0,0,0], [9E9, 9E9, 9E9, 9E9, 9E9, 9E9]];
	VAR robtarget Openhole_2502 := [[444.28, -14.54, 181.4], [-0.031146, 0.70642, 0.707101, 0.002941], [0,0,0,0], [9E9, 9E9, 9E9, 9E9, 9E9, 9E9]];
	VAR robtarget Openhole_2503 := [[442.51, -14.54, 181.48], [-0.037142, 0.706131, 0.70705, 0.008974], [0,0,0,0], [9E9, 9E9, 9E9, 9E9, 9E9, 9E9]];
	VAR robtarget Openhole_2504 := [[441.98, -14.53, 181.5], [-0.038985, 0.706031, 0.707025, 0.010746], [0,0,0,0], [9E9, 9E9, 9E9, 9E9, 9E9, 9E9]];
	VAR robtarget Openhole_2505 := [[440.98, -14.49, 181.55], [-0.042488, 0.705829, 0.706968, 0.013991], [0,0,0,0], [9E9, 9E9, 9E9, 9E9, 9E9, 9E9]];
	VAR robtarget Openhole_2506 := [[439.98, -14.49, 181.59], [-0.045862, 0.705618, 0.706894, 0.017361], [0,0,0,0], [9E9, 9E9, 9E9, 9E9, 9E9, 9E9]];
	VAR robtarget Openhole_2507 := [[439.48, -14.47, 181.61], [-0.047574, 0.705505, 0.706851, 0.019015], [0,0,0,0], [9E9, 9E9, 9E9, 9E9, 9E9, 9E9]];
	VAR robtarget Openhole_2508 := [[438.98, -14.45, 181.64], [-0.049335, 0.705384, 0.706806, 0.020613], [0,0,0,0], [9E9, 9E9, 9E9, 9E9, 9E9, 9E9]];
	VAR robtarget Openhole_2509 := [[438.48, -14.4, 181.66], [-0.051144, 0.705255, 0.70676, 0.02215], [0,0,0,0], [9E9, 9E9, 9E9, 9E9, 9E9, 9E9]];
	VAR robtarget Openhole_2510 := [[433.02, -13.83, 182], [-0.071171, 0.703516, 0.706055, 0.038558], [0,0,0,0], [9E9, 9E9, 9E9, 9E9, 9E9, 9E9]];
	VAR robtarget Openhole_2511 := [[426.54, -13.59, 182.37], [-0.092947, 0.700971, 0.704624, 0.059201], [0,0,0,0], [9E9, 9E9, 9E9, 9E9, 9E9, 9E9]];
	VAR robtarget Openhole_2512 := [[419.55, -13.55, 182.75], [-0.11496, 0.697699, 0.702389, 0.081542], [0,0,0,0], [9E9, 9E9, 9E9, 9E9, 9E9, 9E9]];
	VAR robtarget Openhole_2513 := [[419.05, -13.55, 182.78], [-0.116487, 0.697446, 0.702204, 0.08312], [0,0,0,0], [9E9, 9E9, 9E9, 9E9, 9E9, 9E9]];
	VAR robtarget Openhole_2514 := [[404.07, -13.73, 183.49], [-0.159383, 0.68891, 0.695266, 0.128859], [0,0,0,0], [9E9, 9E9, 9E9, 9E9, 9E9, 9E9]];
	VAR robtarget Openhole_2515 := [[394.35, -14.11, 183.78], [-0.183803, 0.6828, 0.689513, 0.156752], [0,0,0,0], [9E9, 9E9, 9E9, 9E9, 9E9, 9E9]];
	VAR robtarget Openhole_2516 := [[389.35, -14.11, 184.02], [-0.196108, 0.679369, 0.686447, 0.169677], [0,0,0,0], [9E9, 9E9, 9E9, 9E9, 9E9, 9E9]];
	VAR robtarget Openhole_2517 := [[362.35, -14.11, 184.11], [-0.183051, 0.683002, 0.683002, 0.183051], [0,0,0,0], [9E9, 9E9, 9E9, 9E9, 9E9, 9E9]];
	VAR robtarget Openhole_2518 := [[362.35, -15.07, 183.55], [-0.183051, 0.683002, 0.683002, 0.183051], [0,0,0,0], [9E9, 9E9, 9E9, 9E9, 9E9, 9E9]];
	VAR robtarget Openhole_2519 := [[389.35, -15.07, 183.46], [-0.193379, 0.68015, 0.685759, 0.172436], [0,0,0,0], [9E9, 9E9, 9E9, 9E9, 9E9, 9E9]];
	VAR robtarget Openhole_2520 := [[394.35, -15.07, 183.27], [-0.181004, 0.683548, 0.688864, 0.15958], [0,0,0,0], [9E9, 9E9, 9E9, 9E9, 9E9, 9E9]];
	VAR robtarget Openhole_2521 := [[404.04, -14.7, 183.07], [-0.156493, 0.689572, 0.694691, 0.131926], [0,0,0,0], [9E9, 9E9, 9E9, 9E9, 9E9, 9E9]];
	VAR robtarget Openhole_2522 := [[413.54, -14.6, 182.71], [-0.129724, 0.695106, 0.699476, 0.1036], [0,0,0,0], [9E9, 9E9, 9E9, 9E9, 9E9, 9E9]];
	VAR robtarget Openhole_2523 := [[414.03, -14.6, 182.69], [-0.128243, 0.69538, 0.6997, 0.102077], [0,0,0,0], [9E9, 9E9, 9E9, 9E9, 9E9, 9E9]];
	VAR robtarget Openhole_2524 := [[427.52, -14.77, 182.08], [-0.085944, 0.701864, 0.704566, 0.05989], [0,0,0,0], [9E9, 9E9, 9E9, 9E9, 9E9, 9E9]];
	VAR robtarget Openhole_2525 := [[434, -15.12, 181.76], [-0.063635, 0.704238, 0.705995, 0.039635], [0,0,0,0], [9E9, 9E9, 9E9, 9E9, 9E9, 9E9]];
	VAR robtarget Openhole_2526 := [[437.48, -15.49, 181.59], [-0.050841, 0.705277, 0.706503, 0.029224], [0,0,0,0], [9E9, 9E9, 9E9, 9E9, 9E9, 9E9]];
	VAR robtarget Openhole_2527 := [[438.47, -15.58, 181.54], [-0.047221, 0.705528, 0.706623, 0.026161], [0,0,0,0], [9E9, 9E9, 9E9, 9E9, 9E9, 9E9]];
	VAR robtarget Openhole_2528 := [[438.97, -15.61, 181.52], [-0.045463, 0.705644, 0.70668, 0.024562], [0,0,0,0], [9E9, 9E9, 9E9, 9E9, 9E9, 9E9]];
	VAR robtarget Openhole_2529 := [[439.47, -15.62, 181.51], [-0.043738, 0.705753, 0.706735, 0.022924], [0,0,0,0], [9E9, 9E9, 9E9, 9E9, 9E9, 9E9]];
	VAR robtarget Openhole_2530 := [[439.97, -15.62, 181.49], [-0.042046, 0.705856, 0.706788, 0.021247], [0,0,0,0], [9E9, 9E9, 9E9, 9E9, 9E9, 9E9]];
	VAR robtarget Openhole_2531 := [[440.97, -15.59, 181.46], [-0.038784, 0.706042, 0.706884, 0.017763], [0,0,0,0], [9E9, 9E9, 9E9, 9E9, 9E9, 9E9]];
	VAR robtarget Openhole_2532 := [[441.46, -15.51, 181.45], [-0.037417, 0.706116, 0.70693, 0.015802], [0,0,0,0], [9E9, 9E9, 9E9, 9E9, 9E9, 9E9]];
	VAR robtarget Openhole_2533 := [[442.03, -15.46, 181.43], [-0.035664, 0.706207, 0.706974, 0.013687], [0,0,0,0], [9E9, 9E9, 9E9, 9E9, 9E9, 9E9]];
	VAR robtarget Openhole_2534 := [[443.93, -15.46, 181.37], [-0.029254, 0.706501, 0.70707, 0.007244], [0,0,0,0], [9E9, 9E9, 9E9, 9E9, 9E9, 9E9]];
	VAR robtarget Openhole_2535 := [[443.56, -16.48, 181.32], [-0.027038, 0.70659, 0.707005, 0.012004], [0,0,0,0], [9E9, 9E9, 9E9, 9E9, 9E9, 9E9]];
	VAR robtarget Openhole_2536 := [[441.66, -16.48, 181.37], [-0.033449, 0.706315, 0.706866, 0.01844], [0,0,0,0], [9E9, 9E9, 9E9, 9E9, 9E9, 9E9]];
	VAR robtarget Openhole_2537 := [[441.11, -16.58, 181.38], [-0.034973, 0.706241, 0.706806, 0.020616], [0,0,0,0], [9E9, 9E9, 9E9, 9E9, 9E9, 9E9]];
	VAR robtarget Openhole_2538 := [[440.62, -16.69, 181.38], [-0.036238, 0.706178, 0.706744, 0.022644], [0,0,0,0], [9E9, 9E9, 9E9, 9E9, 9E9, 9E9]];
	VAR robtarget Openhole_2539 := [[440.13, -16.73, 181.39], [-0.037783, 0.706097, 0.706683, 0.024463], [0,0,0,0], [9E9, 9E9, 9E9, 9E9, 9E9, 9E9]];
	VAR robtarget Openhole_2540 := [[438.63, -16.79, 181.41], [-0.042626, 0.705821, 0.706482, 0.029716], [0,0,0,0], [9E9, 9E9, 9E9, 9E9, 9E9, 9E9]];
	VAR robtarget Openhole_2541 := [[437.63, -16.79, 181.43], [-0.045966, 0.705611, 0.706332, 0.033094], [0,0,0,0], [9E9, 9E9, 9E9, 9E9, 9E9, 9E9]];
	VAR robtarget Openhole_2542 := [[437.13, -16.79, 181.44], [-0.047645, 0.7055, 0.706252, 0.034767], [0,0,0,0], [9E9, 9E9, 9E9, 9E9, 9E9, 9E9]];
	VAR robtarget Openhole_2543 := [[414.14, -16.27, 182.12], [-0.122624, 0.696393, 0.698955, 0.10706], [0,0,0,0], [9E9, 9E9, 9E9, 9E9, 9E9, 9E9]];
	VAR robtarget Openhole_2544 := [[410.15, -16.25, 182.23], [-0.134474, 0.694202, 0.697025, 0.11898], [0,0,0,0], [9E9, 9E9, 9E9, 9E9, 9E9, 9E9]];
	VAR robtarget Openhole_2545 := [[409.65, -16.25, 182.24], [-0.135922, 0.69392, 0.696771, 0.120456], [0,0,0,0], [9E9, 9E9, 9E9, 9E9, 9E9, 9E9]];
	VAR robtarget Openhole_2546 := [[399.65, -16.42, 182.43], [-0.163226, 0.68801, 0.691146, 0.149389], [0,0,0,0], [9E9, 9E9, 9E9, 9E9, 9E9, 9E9]];
	VAR robtarget Openhole_2547 := [[395.15, -16.63, 182.43], [-0.174413, 0.685259, 0.688291, 0.162034], [0,0,0,0], [9E9, 9E9, 9E9, 9E9, 9E9, 9E9]];
	VAR robtarget Openhole_2548 := [[394.35, -16.66, 182.43], [-0.176391, 0.684753, 0.687771, 0.164228], [0,0,0,0], [9E9, 9E9, 9E9, 9E9, 9E9, 9E9]];
	VAR robtarget Openhole_2549 := [[389.35, -16.66, 182.55], [-0.188882, 0.681413, 0.684603, 0.17697], [0,0,0,0], [9E9, 9E9, 9E9, 9E9, 9E9, 9E9]];
	VAR robtarget Openhole_2550 := [[362.35, -16.66, 182.63], [-0.183051, 0.683002, 0.683002, 0.183051], [0,0,0,0], [9E9, 9E9, 9E9, 9E9, 9E9, 9E9]];
	VAR robtarget Openhole_2551 := [[362.34, -19.81, 180.81], [-0.183051, 0.683002, 0.683002, 0.183051], [0,0,0,0], [9E9, 9E9, 9E9, 9E9, 9E9, 9E9]];
	VAR robtarget Openhole_2552 := [[389.34, -19.81, 180.73], [-0.179931, 0.683831, 0.68222, 0.185945], [0,0,0,0], [9E9, 9E9, 9E9, 9E9, 9E9, 9E9]];
	VAR robtarget Openhole_2553 := [[394.34, -19.81, 180.77], [-0.167212, 0.687052, 0.685508, 0.173431], [0,0,0,0], [9E9, 9E9, 9E9, 9E9, 9E9, 9E9]];
	VAR robtarget Openhole_2554 := [[402.02, -19.48, 180.97], [-0.147569, 0.691537, 0.690549, 0.152127], [0,0,0,0], [9E9, 9E9, 9E9, 9E9, 9E9, 9E9]];
	VAR robtarget Openhole_2555 := [[407.52, -19.42, 181.02], [-0.132198, 0.694639, 0.693801, 0.136528], [0,0,0,0], [9E9, 9E9, 9E9, 9E9, 9E9, 9E9]];
	VAR robtarget Openhole_2556 := [[408.02, -19.42, 181.02], [-0.13075, 0.694913, 0.694082, 0.135095], [0,0,0,0], [9E9, 9E9, 9E9, 9E9, 9E9, 9E9]];
	VAR robtarget Openhole_2557 := [[422.52, -19.62, 181.03], [-0.085986, 0.701859, 0.701103, 0.091945], [0,0,0,0], [9E9, 9E9, 9E9, 9E9, 9E9, 9E9]];
	VAR robtarget Openhole_2558 := [[423.02, -19.61, 181.03], [-0.084398, 0.702052, 0.701309, 0.090364], [0,0,0,0], [9E9, 9E9, 9E9, 9E9, 9E9, 9E9]];
	VAR robtarget Openhole_2559 := [[428.01, -19.47, 181.09], [-0.068776, 0.703754, 0.703236, 0.073885], [0,0,0,0], [9E9, 9E9, 9E9, 9E9, 9E9, 9E9]];
	VAR robtarget Openhole_2560 := [[429.01, -19.4, 181.11], [-0.065747, 0.704044, 0.703592, 0.070419], [0,0,0,0], [9E9, 9E9, 9E9, 9E9, 9E9, 9E9]];
	VAR robtarget Openhole_2561 := [[429.51, -19.35, 181.12], [-0.064274, 0.70418, 0.703767, 0.06864], [0,0,0,0], [9E9, 9E9, 9E9, 9E9, 9E9, 9E9]];
	VAR robtarget Openhole_2562 := [[430.5, -19.24, 181.14], [-0.061392, 0.704437, 0.704111, 0.065016], [0,0,0,0], [9E9, 9E9, 9E9, 9E9, 9E9, 9E9]];
	VAR robtarget Openhole_2563 := [[433.97, -18.76, 181.22], [-0.05156, 0.705224, 0.705195, 0.051961], [0,0,0,0], [9E9, 9E9, 9E9, 9E9, 9E9, 9E9]];
	VAR robtarget Openhole_2564 := [[434.46, -18.67, 181.23], [-0.050202, 0.705322, 0.705334, 0.050042], [0,0,0,0], [9E9, 9E9, 9E9, 9E9, 9E9, 9E9]];
	VAR robtarget Openhole_2565 := [[434.95, -18.6, 181.24], [-0.048801, 0.705421, 0.705465, 0.04815], [0,0,0,0], [9E9, 9E9, 9E9, 9E9, 9E9, 9E9]];
	VAR robtarget Openhole_2566 := [[435.94, -18.42, 181.26], [-0.046137, 0.7056, 0.70572, 0.044256], [0,0,0,0], [9E9, 9E9, 9E9, 9E9, 9E9, 9E9]];
	VAR robtarget Openhole_2567 := [[436.43, -18.34, 181.27], [-0.044755, 0.705689, 0.705838, 0.042338], [0,0,0,0], [9E9, 9E9, 9E9, 9E9, 9E9, 9E9]];
	VAR robtarget Openhole_2568 := [[436.92, -18.24, 181.28], [-0.043443, 0.705771, 0.705954, 0.040367], [0,0,0,0], [9E9, 9E9, 9E9, 9E9, 9E9, 9E9]];
	VAR robtarget Openhole_2569 := [[440.87, -17.63, 181.3], [-0.032234, 0.706372, 0.706665, 0.024978], [0,0,0,0], [9E9, 9E9, 9E9, 9E9, 9E9, 9E9]];
	VAR robtarget Openhole_2570 := [[441.37, -17.54, 181.3], [-0.030859, 0.706433, 0.706732, 0.023023], [0,0,0,0], [9E9, 9E9, 9E9, 9E9, 9E9, 9E9]];
	VAR robtarget Openhole_2571 := [[441.43, -17.55, 181.29], [-0.030612, 0.706444, 0.706738, 0.022838], [0,0,0,0], [9E9, 9E9, 9E9, 9E9, 9E9, 9E9]];
	VAR robtarget Openhole_2572 := [[443.2, -17.55, 181.27], [-0.024612, 0.706678, 0.706907, 0.016825], [0,0,0,0], [9E9, 9E9, 9E9, 9E9, 9E9, 9E9]];
	VAR robtarget Openhole_2573 := [[443.12, -18.53, 181.21], [-0.021549, 0.706778, 0.706811, 0.020446], [0,0,0,0], [9E9, 9E9, 9E9, 9E9, 9E9, 9E9]];
	VAR robtarget Openhole_2574 := [[441.35, -18.53, 181.22], [-0.027553, 0.70657, 0.706612, 0.026454], [0,0,0,0], [9E9, 9E9, 9E9, 9E9, 9E9, 9E9]];
	VAR robtarget Openhole_2575 := [[441.27, -18.53, 181.22], [-0.027817, 0.706559, 0.706602, 0.026709], [0,0,0,0], [9E9, 9E9, 9E9, 9E9, 9E9, 9E9]];
	VAR robtarget Openhole_2576 := [[440.77, -18.58, 181.22], [-0.029333, 0.706498, 0.70653, 0.028556], [0,0,0,0], [9E9, 9E9, 9E9, 9E9, 9E9, 9E9]];
	VAR robtarget Openhole_2577 := [[440.28, -18.68, 181.21], [-0.030665, 0.706442, 0.706447, 0.030537], [0,0,0,0], [9E9, 9E9, 9E9, 9E9, 9E9, 9E9]];
	VAR robtarget Openhole_2578 := [[439.31, -18.93, 181.19], [-0.033091, 0.706332, 0.706258, 0.034642], [0,0,0,0], [9E9, 9E9, 9E9, 9E9, 9E9, 9E9]];
	VAR robtarget Openhole_2579 := [[438.84, -19.07, 181.18], [-0.034211, 0.706279, 0.706152, 0.036742], [0,0,0,0], [9E9, 9E9, 9E9, 9E9, 9E9, 9E9]];
	VAR robtarget Openhole_2580 := [[438.36, -19.23, 181.16], [-0.035256, 0.706227, 0.706037, 0.038878], [0,0,0,0], [9E9, 9E9, 9E9, 9E9, 9E9, 9E9]];
	VAR robtarget Openhole_2581 := [[437.9, -19.41, 181.14], [-0.036204, 0.706179, 0.705914, 0.041055], [0,0,0,0], [9E9, 9E9, 9E9, 9E9, 9E9, 9E9]];
	VAR robtarget Openhole_2582 := [[436.99, -19.83, 181.09], [-0.037844, 0.706093, 0.705641, 0.045501], [0,0,0,0], [9E9, 9E9, 9E9, 9E9, 9E9, 9E9]];
	VAR robtarget Openhole_2583 := [[436.54, -20.05, 181.06], [-0.03863, 0.706051, 0.705494, 0.047731], [0,0,0,0], [9E9, 9E9, 9E9, 9E9, 9E9, 9E9]];
	VAR robtarget Openhole_2584 := [[436.1, -20.28, 181.02], [-0.039324, 0.706012, 0.705338, 0.049987], [0,0,0,0], [9E9, 9E9, 9E9, 9E9, 9E9, 9E9]];
	VAR robtarget Openhole_2585 := [[435.23, -20.76, 180.95], [-0.040619, 0.705939, 0.705002, 0.054514], [0,0,0,0], [9E9, 9E9, 9E9, 9E9, 9E9, 9E9]];
	VAR robtarget Openhole_2586 := [[434.78, -20.99, 180.91], [-0.041336, 0.705898, 0.704826, 0.056752], [0,0,0,0], [9E9, 9E9, 9E9, 9E9, 9E9, 9E9]];
	VAR robtarget Openhole_2587 := [[433.88, -21.41, 180.83], [-0.042933, 0.705802, 0.704457, 0.061156], [0,0,0,0], [9E9, 9E9, 9E9, 9E9, 9E9, 9E9]];
	VAR robtarget Openhole_2588 := [[432.49, -21.97, 180.7], [-0.045698, 0.705629, 0.70387, 0.067585], [0,0,0,0], [9E9, 9E9, 9E9, 9E9, 9E9, 9E9]];
	VAR robtarget Openhole_2589 := [[432.02, -22.13, 180.66], [-0.046706, 0.705563, 0.703665, 0.069679], [0,0,0,0], [9E9, 9E9, 9E9, 9E9, 9E9, 9E9]];
	VAR robtarget Openhole_2590 := [[430.6, -22.59, 180.54], [-0.04989, 0.705345, 0.703026, 0.075853], [0,0,0,0], [9E9, 9E9, 9E9, 9E9, 9E9, 9E9]];
	VAR robtarget Openhole_2591 := [[430.12, -22.73, 180.5], [-0.051014, 0.705264, 0.702806, 0.077868], [0,0,0,0], [9E9, 9E9, 9E9, 9E9, 9E9, 9E9]];
	VAR robtarget Openhole_2592 := [[428.19, -23.21, 180.33], [-0.055797, 0.704902, 0.701894, 0.085704], [0,0,0,0], [9E9, 9E9, 9E9, 9E9, 9E9, 9E9]];
	VAR robtarget Openhole_2593 := [[427.7, -23.31, 180.29], [-0.057062, 0.704801, 0.701659, 0.087606], [0,0,0,0], [9E9, 9E9, 9E9, 9E9, 9E9, 9E9]];
	VAR robtarget Openhole_2594 := [[426.72, -23.49, 180.21], [-0.059677, 0.704584, 0.701183, 0.091334], [0,0,0,0], [9E9, 9E9, 9E9, 9E9, 9E9, 9E9]];
	VAR robtarget Openhole_2595 := [[422.76, -23.95, 179.92], [-0.071027, 0.703531, 0.699218, 0.105328], [0,0,0,0], [9E9, 9E9, 9E9, 9E9, 9E9, 9E9]];
	VAR robtarget Openhole_2596 := [[417.27, -24.13, 179.61], [-0.087871, 0.701626, 0.696375, 0.122727], [0,0,0,0], [9E9, 9E9, 9E9, 9E9, 9E9, 9E9]];
	VAR robtarget Openhole_2597 := [[416.77, -24.13, 179.58], [-0.089429, 0.701429, 0.696108, 0.124233], [0,0,0,0], [9E9, 9E9, 9E9, 9E9, 9E9, 9E9]];
	VAR robtarget Openhole_2598 := [[416.27, -24.13, 179.56], [-0.090993, 0.701228, 0.69584, 0.125723], [0,0,0,0], [9E9, 9E9, 9E9, 9E9, 9E9, 9E9]];
	VAR robtarget Openhole_2599 := [[403.28, -23.96, 178.99], [-0.130383, 0.694982, 0.68825, 0.162211], [0,0,0,0], [9E9, 9E9, 9E9, 9E9, 9E9, 9E9]];
	VAR robtarget Openhole_2600 := [[402.78, -23.96, 178.97], [-0.131802, 0.694714, 0.687929, 0.163565], [0,0,0,0], [9E9, 9E9, 9E9, 9E9, 9E9, 9E9]];
	VAR robtarget Openhole_2601 := [[396.3, -24.14, 178.57], [-0.149272, 0.691171, 0.683526, 0.181086], [0,0,0,0], [9E9, 9E9, 9E9, 9E9, 9E9, 9E9]];
	VAR robtarget Openhole_2602 := [[395.31, -24.2, 178.49], [-0.151784, 0.690624, 0.682808, 0.183773], [0,0,0,0], [9E9, 9E9, 9E9, 9E9, 9E9, 9E9]];
	VAR robtarget Openhole_2603 := [[394.34, -24.22, 178.43], [-0.154312, 0.690064, 0.682133, 0.186263], [0,0,0,0], [9E9, 9E9, 9E9, 9E9, 9E9, 9E9]];
	VAR robtarget Openhole_2604 := [[389.34, -24.22, 178.18], [-0.167348, 0.687019, 0.678686, 0.198458], [0,0,0,0], [9E9, 9E9, 9E9, 9E9, 9E9, 9E9]];
	VAR robtarget Openhole_2605 := [[362.34, -24.22, 178.27], [-0.183051, 0.683002, 0.683002, 0.183051], [0,0,0,0], [9E9, 9E9, 9E9, 9E9, 9E9, 9E9]];
	VAR robtarget Openhole_2606 := [[362.33, -26.32, 177.05], [-0.183051, 0.683002, 0.683002, 0.183051], [0,0,0,0], [9E9, 9E9, 9E9, 9E9, 9E9, 9E9]];
	VAR robtarget Openhole_2607 := [[389.33, -26.32, 176.97], [-0.161335, 0.688455, 0.676922, 0.204394], [0,0,0,0], [9E9, 9E9, 9E9, 9E9, 9E9, 9E9]];
	VAR robtarget Openhole_2608 := [[394.33, -26.32, 177.32], [-0.148148, 0.691413, 0.680442, 0.192352], [0,0,0,0], [9E9, 9E9, 9E9, 9E9, 9E9, 9E9]];
	VAR robtarget Openhole_2609 := [[394.33, -26.32, 177.32], [-0.148166, 0.691409, 0.680437, 0.192367], [0,0,0,0], [9E9, 9E9, 9E9, 9E9, 9E9, 9E9]];
	VAR robtarget Openhole_2610 := [[394.83, -26.28, 177.37], [-0.146928, 0.691673, 0.680819, 0.191013], [0,0,0,0], [9E9, 9E9, 9E9, 9E9, 9E9, 9E9]];
	VAR robtarget Openhole_2611 := [[400.3, -26.08, 177.85], [-0.132399, 0.694601, 0.684725, 0.176499], [0,0,0,0], [9E9, 9E9, 9E9, 9E9, 9E9, 9E9]];
	VAR robtarget Openhole_2612 := [[401.3, -26.08, 177.92], [-0.12959, 0.69513, 0.685398, 0.173868], [0,0,0,0], [9E9, 9E9, 9E9, 9E9, 9E9, 9E9]];
	VAR robtarget Openhole_2613 := [[401.8, -26.08, 177.95], [-0.128169, 0.695394, 0.68573, 0.172552], [0,0,0,0], [9E9, 9E9, 9E9, 9E9, 9E9, 9E9]];
	VAR robtarget Openhole_2614 := [[416.77, -26.42, 178.86], [-0.082092, 0.702325, 0.694769, 0.131513], [0,0,0,0], [9E9, 9E9, 9E9, 9E9, 9E9, 9E9]];
	VAR robtarget Openhole_2615 := [[417.27, -26.42, 178.9], [-0.080523, 0.702507, 0.69505, 0.130024], [0,0,0,0], [9E9, 9E9, 9E9, 9E9, 9E9, 9E9]];
	VAR robtarget Openhole_2616 := [[422.25, -26.24, 179.3], [-0.065184, 0.704096, 0.697801, 0.114339], [0,0,0,0], [9E9, 9E9, 9E9, 9E9, 9E9, 9E9]];
	VAR robtarget Openhole_2617 := [[426.2, -25.8, 179.67], [-0.053755, 0.705061, 0.699923, 0.100537], [0,0,0,0], [9E9, 9E9, 9E9, 9E9, 9E9, 9E9]];
	VAR robtarget Openhole_2618 := [[426.69, -25.72, 179.72], [-0.052405, 0.705162, 0.700182, 0.098721], [0,0,0,0], [9E9, 9E9, 9E9, 9E9, 9E9, 9E9]];
	VAR robtarget Openhole_2619 := [[428.64, -25.31, 179.93], [-0.047319, 0.705522, 0.701202, 0.091187], [0,0,0,0], [9E9, 9E9, 9E9, 9E9, 9E9, 9E9]];
	VAR robtarget Openhole_2620 := [[431.04, -24.65, 180.19], [-0.041591, 0.705883, 0.702422, 0.081259], [0,0,0,0], [9E9, 9E9, 9E9, 9E9, 9E9, 9E9]];
	VAR robtarget Openhole_2621 := [[431.98, -24.33, 180.3], [-0.039516, 0.706002, 0.702887, 0.077136], [0,0,0,0], [9E9, 9E9, 9E9, 9E9, 9E9, 9E9]];
	VAR robtarget Openhole_2622 := [[432.44, -24.15, 180.35], [-0.038558, 0.706055, 0.703115, 0.075029], [0,0,0,0], [9E9, 9E9, 9E9, 9E9, 9E9, 9E9]];
	VAR robtarget Openhole_2623 := [[433.36, -23.77, 180.45], [-0.036771, 0.70615, 0.703559, 0.070746], [0,0,0,0], [9E9, 9E9, 9E9, 9E9, 9E9, 9E9]];
	VAR robtarget Openhole_2624 := [[434.26, -23.35, 180.55], [-0.035166, 0.706232, 0.703985, 0.066374], [0,0,0,0], [9E9, 9E9, 9E9, 9E9, 9E9, 9E9]];
	VAR robtarget Openhole_2625 := [[435.15, -22.9, 180.65], [-0.0337, 0.706303, 0.704389, 0.061935], [0,0,0,0], [9E9, 9E9, 9E9, 9E9, 9E9, 9E9]];
	VAR robtarget Openhole_2626 := [[436.02, -22.42, 180.75], [-0.032387, 0.706365, 0.704771, 0.057432], [0,0,0,0], [9E9, 9E9, 9E9, 9E9, 9E9, 9E9]];
	VAR robtarget Openhole_2627 := [[436.45, -22.16, 180.79], [-0.031789, 0.706392, 0.704952, 0.055158], [0,0,0,0], [9E9, 9E9, 9E9, 9E9, 9E9, 9E9]];
	VAR robtarget Openhole_2628 := [[438.54, -20.81, 181], [-0.029306, 0.706499, 0.705761, 0.043609], [0,0,0,0], [9E9, 9E9, 9E9, 9E9, 9E9, 9E9]];
	VAR robtarget Openhole_2629 := [[438.97, -20.55, 181.03], [-0.028735, 0.706523, 0.705899, 0.041305], [0,0,0,0], [9E9, 9E9, 9E9, 9E9, 9E9, 9E9]];
	VAR robtarget Openhole_2630 := [[439.41, -20.32, 181.06], [-0.028035, 0.706551, 0.706029, 0.039033], [0,0,0,0], [9E9, 9E9, 9E9, 9E9, 9E9, 9E9]];
	VAR robtarget Openhole_2631 := [[439.86, -20.1, 181.08], [-0.027261, 0.706581, 0.706149, 0.036783], [0,0,0,0], [9E9, 9E9, 9E9, 9E9, 9E9, 9E9]];
	VAR robtarget Openhole_2632 := [[440.31, -19.89, 181.11], [-0.02644, 0.706612, 0.706262, 0.034545], [0,0,0,0], [9E9, 9E9, 9E9, 9E9, 9E9, 9E9]];
	VAR robtarget Openhole_2633 := [[440.77, -19.7, 181.13], [-0.025561, 0.706645, 0.706367, 0.032328], [0,0,0,0], [9E9, 9E9, 9E9, 9E9, 9E9, 9E9]];
	VAR robtarget Openhole_2634 := [[441.39, -19.52, 181.14], [-0.024072, 0.706697, 0.706484, 0.029663], [0,0,0,0], [9E9, 9E9, 9E9, 9E9, 9E9, 9E9]];
	VAR robtarget Openhole_2635 := [[443.53, -19.52, 181.15], [-0.016818, 0.706907, 0.706751, 0.022415], [0,0,0,0], [9E9, 9E9, 9E9, 9E9, 9E9, 9E9]];
	VAR robtarget Openhole_2636 := [[443.72, -20.63, 181.09], [-0.012388, 0.706998, 0.706646, 0.025529], [0,0,0,0], [9E9, 9E9, 9E9, 9E9, 9E9, 9E9]];
	VAR robtarget Openhole_2637 := [[441.58, -20.63, 181.06], [-0.019649, 0.706834, 0.706347, 0.032773], [0,0,0,0], [9E9, 9E9, 9E9, 9E9, 9E9, 9E9]];
	VAR robtarget Openhole_2638 := [[440.79, -20.96, 181.02], [-0.021213, 0.706789, 0.706161, 0.036558], [0,0,0,0], [9E9, 9E9, 9E9, 9E9, 9E9, 9E9]];
	VAR robtarget Openhole_2639 := [[438.24, -22.52, 180.81], [-0.024562, 0.70668, 0.705308, 0.050399], [0,0,0,0], [9E9, 9E9, 9E9, 9E9, 9E9, 9E9]];
	VAR robtarget Openhole_2640 := [[436.52, -23.52, 180.63], [-0.026989, 0.706592, 0.704599, 0.059506], [0,0,0,0], [9E9, 9E9, 9E9, 9E9, 9E9, 9E9]];
	VAR robtarget Openhole_2641 := [[435.19, -24.2, 180.48], [-0.029174, 0.706505, 0.704003, 0.066185], [0,0,0,0], [9E9, 9E9, 9E9, 9E9, 9E9, 9E9]];
	VAR robtarget Openhole_2642 := [[434.29, -24.62, 180.37], [-0.030797, 0.706436, 0.703578, 0.070559], [0,0,0,0], [9E9, 9E9, 9E9, 9E9, 9E9, 9E9]];
	VAR robtarget Openhole_2643 := [[433.83, -24.82, 180.32], [-0.031666, 0.706397, 0.703358, 0.072717], [0,0,0,0], [9E9, 9E9, 9E9, 9E9, 9E9, 9E9]];
	VAR robtarget Openhole_2644 := [[433.37, -25.01, 180.26], [-0.032575, 0.706356, 0.703134, 0.074854], [0,0,0,0], [9E9, 9E9, 9E9, 9E9, 9E9, 9E9]];
	VAR robtarget Openhole_2645 := [[432.91, -25.19, 180.21], [-0.03353, 0.706311, 0.702906, 0.076966], [0,0,0,0], [9E9, 9E9, 9E9, 9E9, 9E9, 9E9]];
	VAR robtarget Openhole_2646 := [[429.59, -26.22, 179.81], [-0.041164, 0.705908, 0.701208, 0.091144], [0,0,0,0], [9E9, 9E9, 9E9, 9E9, 9E9, 9E9]];
	VAR robtarget Openhole_2647 := [[426.18, -26.93, 179.42], [-0.050087, 0.705331, 0.699374, 0.104291], [0,0,0,0], [9E9, 9E9, 9E9, 9E9, 9E9, 9E9]];
	VAR robtarget Openhole_2648 := [[422.23, -27.36, 179.01], [-0.061591, 0.704419, 0.697192, 0.117996], [0,0,0,0], [9E9, 9E9, 9E9, 9E9, 9E9, 9E9]];
	VAR robtarget Openhole_2649 := [[416.76, -27.54, 178.51], [-0.078539, 0.702732, 0.694083, 0.13509], [0,0,0,0], [9E9, 9E9, 9E9, 9E9, 9E9, 9E9]];
	VAR robtarget Openhole_2650 := [[416.26, -27.54, 178.47], [-0.080118, 0.702553, 0.693795, 0.136558], [0,0,0,0], [9E9, 9E9, 9E9, 9E9, 9E9, 9E9]];
	VAR robtarget Openhole_2651 := [[405.79, -27.19, 177.76], [-0.113188, 0.697989, 0.687539, 0.165197], [0,0,0,0], [9E9, 9E9, 9E9, 9E9, 9E9, 9E9]];
	VAR robtarget Openhole_2652 := [[399.8, -27.04, 177.36], [-0.130934, 0.694879, 0.683649, 0.180621], [0,0,0,0], [9E9, 9E9, 9E9, 9E9, 9E9, 9E9]];
	VAR robtarget Openhole_2653 := [[399.31, -27.04, 177.32], [-0.132334, 0.694613, 0.683307, 0.181911], [0,0,0,0], [9E9, 9E9, 9E9, 9E9, 9E9, 9E9]];
	VAR robtarget Openhole_2654 := [[394.26, -27.21, 176.85], [-0.145777, 0.691917, 0.679665, 0.195078], [0,0,0,0], [9E9, 9E9, 9E9, 9E9, 9E9, 9E9]];
	VAR robtarget Openhole_2655 := [[389.33, -27.21, 176.46], [-0.158818, 0.689041, 0.676169, 0.206871], [0,0,0,0], [9E9, 9E9, 9E9, 9E9, 9E9, 9E9]];
	VAR robtarget Openhole_2656 := [[362.33, -27.21, 176.54], [-0.183051, 0.683002, 0.683002, 0.183051], [0,0,0,0], [9E9, 9E9, 9E9, 9E9, 9E9, 9E9]];
	VAR robtarget Openhole_2657 := [[362.33, -28.09, 176.03], [-0.183051, 0.683002, 0.683002, 0.183051], [0,0,0,0], [9E9, 9E9, 9E9, 9E9, 9E9, 9E9]];
	VAR robtarget Openhole_2658 := [[389.33, -28.09, 175.95], [-0.156297, 0.689617, 0.675406, 0.209347], [0,0,0,0], [9E9, 9E9, 9E9, 9E9, 9E9, 9E9]];
	VAR robtarget Openhole_2659 := [[394.33, -28.09, 176.38], [-0.142986, 0.692499, 0.678985, 0.197432], [0,0,0,0], [9E9, 9E9, 9E9, 9E9, 9E9, 9E9]];
	VAR robtarget Openhole_2660 := [[395.18, -28.08, 176.46], [-0.140689, 0.692969, 0.679588, 0.195346], [0,0,0,0], [9E9, 9E9, 9E9, 9E9, 9E9, 9E9]];
	VAR robtarget Openhole_2661 := [[398.16, -28.02, 176.75], [-0.13262, 0.694559, 0.681738, 0.187704], [0,0,0,0], [9E9, 9E9, 9E9, 9E9, 9E9, 9E9]];
	VAR robtarget Openhole_2662 := [[398.66, -28.02, 176.79], [-0.131217, 0.694825, 0.682084, 0.186445], [0,0,0,0], [9E9, 9E9, 9E9, 9E9, 9E9, 9E9]];
	VAR robtarget Openhole_2663 := [[405.64, -28.29, 177.29], [-0.110267, 0.698456, 0.686633, 0.168925], [0,0,0,0], [9E9, 9E9, 9E9, 9E9, 9E9, 9E9]];
	VAR robtarget Openhole_2664 := [[415.1, -28.72, 177.99], [-0.079974, 0.70257, 0.692353, 0.14369], [0,0,0,0], [9E9, 9E9, 9E9, 9E9, 9E9, 9E9]];
	VAR robtarget Openhole_2665 := [[417.09, -28.75, 178.16], [-0.073602, 0.703266, 0.693526, 0.137921], [0,0,0,0], [9E9, 9E9, 9E9, 9E9, 9E9, 9E9]];
	VAR robtarget Openhole_2666 := [[417.59, -28.74, 178.21], [-0.072024, 0.703429, 0.693818, 0.136441], [0,0,0,0], [9E9, 9E9, 9E9, 9E9, 9E9, 9E9]];
	VAR robtarget Openhole_2667 := [[423.06, -28.53, 178.78], [-0.055087, 0.704958, 0.696981, 0.119238], [0,0,0,0], [9E9, 9E9, 9E9, 9E9, 9E9, 9E9]];
	VAR robtarget Openhole_2668 := [[427, -28.06, 179.24], [-0.043667, 0.705757, 0.699204, 0.105419], [0,0,0,0], [9E9, 9E9, 9E9, 9E9, 9E9, 9E9]];
	VAR robtarget Openhole_2669 := [[430.4, -27.35, 179.66], [-0.034713, 0.706254, 0.701062, 0.092259], [0,0,0,0], [9E9, 9E9, 9E9, 9E9, 9E9, 9E9]];
	VAR robtarget Openhole_2670 := [[432.32, -26.83, 179.9], [-0.03004, 0.706468, 0.702059, 0.084342], [0,0,0,0], [9E9, 9E9, 9E9, 9E9, 9E9, 9E9]];
	VAR robtarget Openhole_2671 := [[433.73, -26.37, 180.08], [-0.026801, 0.706599, 0.702769, 0.078206], [0,0,0,0], [9E9, 9E9, 9E9, 9E9, 9E9, 9E9]];
	VAR robtarget Openhole_2672 := [[434.67, -26.03, 180.19], [-0.024809, 0.706671, 0.703223, 0.07401], [0,0,0,0], [9E9, 9E9, 9E9, 9E9, 9E9, 9E9]];
	VAR robtarget Openhole_2673 := [[437.86, -24.65, 180.56], [-0.018666, 0.70686, 0.704656, 0.058823], [0,0,0,0], [9E9, 9E9, 9E9, 9E9, 9E9, 9E9]];
	VAR robtarget Openhole_2674 := [[438.31, -24.43, 180.61], [-0.017906, 0.70688, 0.704838, 0.056592], [0,0,0,0], [9E9, 9E9, 9E9, 9E9, 9E9, 9E9]];
	VAR robtarget Openhole_2675 := [[439.62, -23.72, 180.74], [-0.015838, 0.706929, 0.70535, 0.049812], [0,0,0,0], [9E9, 9E9, 9E9, 9E9, 9E9, 9E9]];
	VAR robtarget Openhole_2676 := [[440.05, -23.46, 180.78], [-0.015254, 0.706942, 0.705509, 0.047515], [0,0,0,0], [9E9, 9E9, 9E9, 9E9, 9E9, 9E9]];
	VAR robtarget Openhole_2677 := [[441.31, -22.66, 180.9], [-0.013692, 0.706974, 0.705943, 0.040561], [0,0,0,0], [9E9, 9E9, 9E9, 9E9, 9E9, 9E9]];
	VAR robtarget Openhole_2678 := [[442.15, -22.2, 180.96], [-0.0124, 0.706998, 0.706181, 0.036169], [0,0,0,0], [9E9, 9E9, 9E9, 9E9, 9E9, 9E9]];
	VAR robtarget Openhole_2679 := [[443.96, -22.2, 181.02], [-0.006271, 0.707079, 0.706467, 0.030067], [0,0,0,0], [9E9, 9E9, 9E9, 9E9, 9E9, 9E9]];
	VAR robtarget Openhole_2680 := [[445.39, -24.26, 180.98], [0.005584, 0.707085, 0.706375, 0.032169], [0,0,0,0], [9E9, 9E9, 9E9, 9E9, 9E9, 9E9]];
	VAR robtarget Openhole_2681 := [[443.59, -24.26, 180.89], [-0.000557, 0.707107, 0.70607, 0.038277], [0,0,0,0], [9E9, 9E9, 9E9, 9E9, 9E9, 9E9]];
	VAR robtarget Openhole_2682 := [[442.83, -24.81, 180.82], [-0.00127, 0.707106, 0.705816, 0.04271], [0,0,0,0], [9E9, 9E9, 9E9, 9E9, 9E9, 9E9]];
	VAR robtarget Openhole_2683 := [[441.94, -25.27, 180.74], [-0.002736, 0.707101, 0.705527, 0.047237], [0,0,0,0], [9E9, 9E9, 9E9, 9E9, 9E9, 9E9]];
	VAR robtarget Openhole_2684 := [[441.49, -25.47, 180.69], [-0.003607, 0.707098, 0.705376, 0.049447], [0,0,0,0], [9E9, 9E9, 9E9, 9E9, 9E9, 9E9]];
	VAR robtarget Openhole_2685 := [[441.02, -25.65, 180.65], [-0.004583, 0.707092, 0.705221, 0.05161], [0,0,0,0], [9E9, 9E9, 9E9, 9E9, 9E9, 9E9]];
	VAR robtarget Openhole_2686 := [[439.61, -26.14, 180.52], [-0.007693, 0.707065, 0.704724, 0.057998], [0,0,0,0], [9E9, 9E9, 9E9, 9E9, 9E9, 9E9]];
	VAR robtarget Openhole_2687 := [[433.43, -28.02, 179.8], [-0.022295, 0.706755, 0.702019, 0.084671], [0,0,0,0], [9E9, 9E9, 9E9, 9E9, 9E9, 9E9]];
	VAR robtarget Openhole_2688 := [[429.08, -29, 179.24], [-0.033663, 0.706305, 0.699725, 0.101904], [0,0,0,0], [9E9, 9E9, 9E9, 9E9, 9E9, 9E9]];
	VAR robtarget Openhole_2689 := [[424.66, -29.62, 178.66], [-0.04626, 0.705592, 0.697224, 0.117809], [0,0,0,0], [9E9, 9E9, 9E9, 9E9, 9E9, 9E9]];
	VAR robtarget Openhole_2690 := [[420.2, -29.9, 178.13], [-0.059909, 0.704564, 0.694616, 0.132318], [0,0,0,0], [9E9, 9E9, 9E9, 9E9, 9E9, 9E9]];
	VAR robtarget Openhole_2691 := [[417.72, -29.94, 177.86], [-0.067779, 0.703851, 0.693139, 0.13985], [0,0,0,0], [9E9, 9E9, 9E9, 9E9, 9E9, 9E9]];
	VAR robtarget Openhole_2692 := [[417.22, -29.94, 177.81], [-0.069375, 0.703695, 0.692843, 0.14131], [0,0,0,0], [9E9, 9E9, 9E9, 9E9, 9E9, 9E9]];
	VAR robtarget Openhole_2693 := [[410.75, -29.69, 177.22], [-0.090446, 0.701298, 0.688969, 0.159128], [0,0,0,0], [9E9, 9E9, 9E9, 9E9, 9E9, 9E9]];
	VAR robtarget Openhole_2694 := [[399.3, -28.99, 176.39], [-0.12651, 0.695698, 0.681758, 0.187632], [0,0,0,0], [9E9, 9E9, 9E9, 9E9, 9E9, 9E9]];
	VAR robtarget Openhole_2695 := [[396.81, -28.94, 176.17], [-0.133641, 0.694363, 0.680039, 0.193772], [0,0,0,0], [9E9, 9E9, 9E9, 9E9, 9E9, 9E9]];
	VAR robtarget Openhole_2696 := [[396.32, -28.94, 176.12], [-0.135017, 0.694097, 0.679684, 0.195012], [0,0,0,0], [9E9, 9E9, 9E9, 9E9, 9E9, 9E9]];
	VAR robtarget Openhole_2697 := [[394.82, -28.97, 175.97], [-0.139062, 0.693298, 0.678602, 0.198746], [0,0,0,0], [9E9, 9E9, 9E9, 9E9, 9E9, 9E9]];
	VAR robtarget Openhole_2698 := [[394.3, -28.99, 175.9], [-0.140417, 0.693025, 0.678209, 0.200082], [0,0,0,0], [9E9, 9E9, 9E9, 9E9, 9E9, 9E9]];
	VAR robtarget Openhole_2699 := [[389.33, -28.99, 175.43], [-0.153721, 0.690195, 0.674619, 0.211871], [0,0,0,0], [9E9, 9E9, 9E9, 9E9, 9E9, 9E9]];
	VAR robtarget Openhole_2700 := [[362.33, -28.99, 175.51], [-0.183051, 0.683002, 0.683002, 0.183051], [0,0,0,0], [9E9, 9E9, 9E9, 9E9, 9E9, 9E9]];
	VAR robtarget Openhole_2701 := [[362.32, -30.66, 174.55], [-0.183051, 0.683002, 0.683002, 0.183051], [0,0,0,0], [9E9, 9E9, 9E9, 9E9, 9E9, 9E9]];
	VAR robtarget Openhole_2702 := [[374.32, -30.66, 174.51], [-0.183051, 0.683002, 0.683002, 0.183051], [0,0,0,0], [9E9, 9E9, 9E9, 9E9, 9E9, 9E9]];
	VAR robtarget Openhole_2703 := [[389.32, -30.66, 174.46], [-0.14896, 0.691239, 0.67314, 0.216524], [0,0,0,0], [9E9, 9E9, 9E9, 9E9, 9E9, 9E9]];
	VAR robtarget Openhole_2704 := [[394.83, -30.66, 175.08], [-0.134068, 0.694281, 0.677163, 0.203593], [0,0,0,0], [9E9, 9E9, 9E9, 9E9, 9E9, 9E9]];
	VAR robtarget Openhole_2705 := [[399.31, -30.93, 175.45], [-0.12068, 0.696733, 0.680167, 0.193321], [0,0,0,0], [9E9, 9E9, 9E9, 9E9, 9E9, 9E9]];
	VAR robtarget Openhole_2706 := [[410.71, -32.09, 176.32], [-0.083051, 0.702213, 0.6872, 0.1666], [0,0,0,0], [9E9, 9E9, 9E9, 9E9, 9E9, 9E9]];
	VAR robtarget Openhole_2707 := [[417.16, -32.5, 177.01], [-0.061384, 0.704437, 0.691121, 0.149503], [0,0,0,0], [9E9, 9E9, 9E9, 9E9, 9E9, 9E9]];
	VAR robtarget Openhole_2708 := [[419.64, -32.54, 177.32], [-0.053228, 0.705101, 0.692632, 0.14234], [0,0,0,0], [9E9, 9E9, 9E9, 9E9, 9E9, 9E9]];
	VAR robtarget Openhole_2709 := [[420.14, -32.54, 177.38], [-0.051616, 0.70522, 0.692934, 0.140865], [0,0,0,0], [9E9, 9E9, 9E9, 9E9, 9E9, 9E9]];
	VAR robtarget Openhole_2710 := [[425.09, -32.35, 178.07], [-0.035944, 0.706193, 0.695921, 0.125276], [0,0,0,0], [9E9, 9E9, 9E9, 9E9, 9E9, 9E9]];
	VAR robtarget Openhole_2711 := [[430.5, -31.78, 178.87], [-0.019701, 0.706832, 0.699042, 0.106492], [0,0,0,0], [9E9, 9E9, 9E9, 9E9, 9E9, 9E9]];
	VAR robtarget Openhole_2712 := [[437.38, -30.92, 179.81], [0.000748, 0.707106, 0.70241, 0.081367], [0,0,0,0], [9E9, 9E9, 9E9, 9E9, 9E9, 9E9]];
	VAR robtarget Openhole_2713 := [[438.37, -30.84, 179.93], [0.003833, 0.707096, 0.702811, 0.077826], [0,0,0,0], [9E9, 9E9, 9E9, 9E9, 9E9, 9E9]];
	VAR robtarget Openhole_2714 := [[439.36, -30.78, 180.05], [0.007019, 0.707072, 0.703187, 0.074355], [0,0,0,0], [9E9, 9E9, 9E9, 9E9, 9E9, 9E9]];
	VAR robtarget Openhole_2715 := [[440.85, -30.75, 180.22], [0.011977, 0.707005, 0.703704, 0.069285], [0,0,0,0], [9E9, 9E9, 9E9, 9E9, 9E9, 9E9]];
	VAR robtarget Openhole_2716 := [[441.35, -30.75, 180.28], [0.013673, 0.706975, 0.703865, 0.067629], [0,0,0,0], [9E9, 9E9, 9E9, 9E9, 9E9, 9E9]];
	VAR robtarget Openhole_2717 := [[445.32, -30.96, 180.72], [0.027916, 0.706556, 0.704963, 0.055016], [0,0,0,0], [9E9, 9E9, 9E9, 9E9, 9E9, 9E9]];
	VAR robtarget Openhole_2718 := [[449.27, -31.31, 181.17], [0.042573, 0.705824, 0.70581, 0.042811], [0,0,0,0], [9E9, 9E9, 9E9, 9E9, 9E9, 9E9]];
	VAR robtarget Openhole_2719 := [[449.77, -31.34, 181.23], [0.044332, 0.705716, 0.705905, 0.041201], [0,0,0,0], [9E9, 9E9, 9E9, 9E9, 9E9, 9E9]];
	VAR robtarget Openhole_2720 := [[450.27, -31.35, 181.29], [0.046063, 0.705605, 0.705999, 0.039559], [0,0,0,0], [9E9, 9E9, 9E9, 9E9, 9E9, 9E9]];
	VAR robtarget Openhole_2721 := [[450.76, -31.35, 181.35], [0.047744, 0.705493, 0.706092, 0.037871], [0,0,0,0], [9E9, 9E9, 9E9, 9E9, 9E9, 9E9]];
	VAR robtarget Openhole_2722 := [[451.76, -31.32, 181.47], [0.05098, 0.705267, 0.706271, 0.03437], [0,0,0,0], [9E9, 9E9, 9E9, 9E9, 9E9, 9E9]];
	VAR robtarget Openhole_2723 := [[452.75, -31.23, 181.58], [0.054038, 0.705039, 0.70644, 0.030711], [0,0,0,0], [9E9, 9E9, 9E9, 9E9, 9E9, 9E9]];
	VAR robtarget Openhole_2724 := [[453.73, -31.11, 181.69], [0.056957, 0.704809, 0.706593, 0.02694], [0,0,0,0], [9E9, 9E9, 9E9, 9E9, 9E9, 9E9]];
	VAR robtarget Openhole_2725 := [[461.6, -29.87, 182.46], [0.079027, 0.702677, 0.707095, -0.004036], [0,0,0,0], [9E9, 9E9, 9E9, 9E9, 9E9, 9E9]];
	VAR robtarget Openhole_2726 := [[470.52, -29.03, 183.22], [0.105055, 0.699259, 0.706141, -0.036943], [0,0,0,0], [9E9, 9E9, 9E9, 9E9, 9E9, 9E9]];
	VAR robtarget Openhole_2727 := [[482.96, -28.21, 184.15], [0.140336, 0.693041, 0.702565, -0.080019], [0,0,0,0], [9E9, 9E9, 9E9, 9E9, 9E9, 9E9]];
	VAR robtarget Openhole_2728 := [[502.4, -27.36, 185.44], [0.190539, 0.680952, 0.693077, -0.140156], [0,0,0,0], [9E9, 9E9, 9E9, 9E9, 9E9, 9E9]];
	VAR robtarget Openhole_2729 := [[504.36, -27.26, 185.54], [0.195094, 0.679661, 0.691914, -0.145793], [0,0,0,0], [9E9, 9E9, 9E9, 9E9, 9E9, 9E9]];
	VAR robtarget Openhole_2730 := [[509.36, -27.26, 185.94], [0.183051, 0.683002, 0.683002, -0.183051], [0,0,0,0], [9E9, 9E9, 9E9, 9E9, 9E9, 9E9]];
	VAR robtarget Openhole_2731 := [[536.36, -27.26, 185.85], [0.183051, 0.683002, 0.683002, -0.183051], [0,0,0,0], [9E9, 9E9, 9E9, 9E9, 9E9, 9E9]];
	VAR robtarget Openhole_2732 := [[536.36, -28.38, 186.5], [0.183051, 0.683002, 0.683002, -0.183051], [0,0,0,0], [9E9, 9E9, 9E9, 9E9, 9E9, 9E9]];
	VAR robtarget Openhole_2733 := [[509.36, -28.38, 186.59], [0.183051, 0.683002, 0.683002, -0.183051], [0,0,0,0], [9E9, 9E9, 9E9, 9E9, 9E9, 9E9]];
	VAR robtarget Openhole_2734 := [[504.36, -28.38, 186.14], [0.198308, 0.67873, 0.692596, -0.142516], [0,0,0,0], [9E9, 9E9, 9E9, 9E9, 9E9, 9E9]];
	VAR robtarget Openhole_2735 := [[483.56, -29.45, 184.61], [0.145986, 0.691873, 0.702796, -0.077956], [0,0,0,0], [9E9, 9E9, 9E9, 9E9, 9E9, 9E9]];
	VAR robtarget Openhole_2736 := [[473.63, -30.27, 183.81], [0.118782, 0.697059, 0.705787, -0.04319], [0,0,0,0], [9E9, 9E9, 9E9, 9E9, 9E9, 9E9]];
	VAR robtarget Openhole_2737 := [[466.21, -31.16, 183.15], [0.098292, 0.700242, 0.706939, -0.01541], [0,0,0,0], [9E9, 9E9, 9E9, 9E9, 9E9, 9E9]];
	VAR robtarget Openhole_2738 := [[460.33, -32.16, 182.57], [0.082415, 0.702287, 0.707062, 0.00792], [0,0,0,0], [9E9, 9E9, 9E9, 9E9, 9E9, 9E9]];
	VAR robtarget Openhole_2739 := [[452.59, -33.96, 181.65], [0.062608, 0.70433, 0.705954, 0.040368], [0,0,0,0], [9E9, 9E9, 9E9, 9E9, 9E9, 9E9]];
	VAR robtarget Openhole_2740 := [[452.1, -34.05, 181.58], [0.061234, 0.70445, 0.70584, 0.042306], [0,0,0,0], [9E9, 9E9, 9E9, 9E9, 9E9, 9E9]];
	VAR robtarget Openhole_2741 := [[451.61, -34.11, 181.51], [0.059801, 0.704573, 0.705724, 0.044202], [0,0,0,0], [9E9, 9E9, 9E9, 9E9, 9E9, 9E9]];
	VAR robtarget Openhole_2742 := [[451.12, -34.17, 181.44], [0.058317, 0.704698, 0.705605, 0.046054], [0,0,0,0], [9E9, 9E9, 9E9, 9E9, 9E9, 9E9]];
	VAR robtarget Openhole_2743 := [[450.62, -34.2, 181.37], [0.056756, 0.704825, 0.705486, 0.047844], [0,0,0,0], [9E9, 9E9, 9E9, 9E9, 9E9, 9E9]];
	VAR robtarget Openhole_2744 := [[450.13, -34.22, 181.3], [0.055148, 0.704953, 0.705366, 0.049589], [0,0,0,0], [9E9, 9E9, 9E9, 9E9, 9E9, 9E9]];
	VAR robtarget Openhole_2745 := [[449.64, -34.22, 181.22], [0.053471, 0.705082, 0.705246, 0.051268], [0,0,0,0], [9E9, 9E9, 9E9, 9E9, 9E9, 9E9]];
	VAR robtarget Openhole_2746 := [[449.14, -34.2, 181.15], [0.051749, 0.705211, 0.705125, 0.052901], [0,0,0,0], [9E9, 9E9, 9E9, 9E9, 9E9, 9E9]];
	VAR robtarget Openhole_2747 := [[448.65, -34.17, 181.08], [0.049959, 0.70534, 0.705006, 0.054462], [0,0,0,0], [9E9, 9E9, 9E9, 9E9, 9E9, 9E9]];
	VAR robtarget Openhole_2748 := [[448.15, -34.12, 181.01], [0.048126, 0.705467, 0.704888, 0.055969], [0,0,0,0], [9E9, 9E9, 9E9, 9E9, 9E9, 9E9]];
	VAR robtarget Openhole_2749 := [[447.66, -34.06, 180.94], [0.046252, 0.705592, 0.704771, 0.057426], [0,0,0,0], [9E9, 9E9, 9E9, 9E9, 9E9, 9E9]];
	VAR robtarget Openhole_2750 := [[442.77, -33.27, 180.28], [0.026943, 0.706593, 0.703508, 0.071252], [0,0,0,0], [9E9, 9E9, 9E9, 9E9, 9E9, 9E9]];
	VAR robtarget Openhole_2751 := [[439.31, -33.03, 179.83], [0.014332, 0.706962, 0.70234, 0.081969], [0,0,0,0], [9E9, 9E9, 9E9, 9E9, 9E9, 9E9]];
	VAR robtarget Openhole_2752 := [[438.32, -33.02, 179.7], [0.010914, 0.707023, 0.701955, 0.085201], [0,0,0,0], [9E9, 9E9, 9E9, 9E9, 9E9, 9E9]];
	VAR robtarget Openhole_2753 := [[437.82, -33.02, 179.63], [0.009243, 0.707046, 0.701753, 0.08685], [0,0,0,0], [9E9, 9E9, 9E9, 9E9, 9E9, 9E9]];
	VAR robtarget Openhole_2754 := [[433.38, -33.3, 178.99], [-0.004978, 0.707089, 0.699682, 0.102204], [0,0,0,0], [9E9, 9E9, 9E9, 9E9, 9E9, 9E9]];
	VAR robtarget Openhole_2755 := [[425.51, -33.98, 177.75], [-0.029265, 0.706501, 0.695204, 0.129195], [0,0,0,0], [9E9, 9E9, 9E9, 9E9, 9E9, 9E9]];
	VAR robtarget Openhole_2756 := [[421.06, -34.1, 177.08], [-0.043599, 0.705761, 0.692487, 0.143044], [0,0,0,0], [9E9, 9E9, 9E9, 9E9, 9E9, 9E9]];
	VAR robtarget Openhole_2757 := [[420.56, -34.09, 177.01], [-0.045228, 0.705659, 0.692182, 0.144512], [0,0,0,0], [9E9, 9E9, 9E9, 9E9, 9E9, 9E9]];
	VAR robtarget Openhole_2758 := [[415.12, -33.89, 176.29], [-0.063542, 0.704246, 0.688831, 0.159723], [0,0,0,0], [9E9, 9E9, 9E9, 9E9, 9E9, 9E9]];
	VAR robtarget Openhole_2759 := [[408.68, -33.3, 175.6], [-0.085596, 0.701907, 0.684898, 0.175827], [0,0,0,0], [9E9, 9E9, 9E9, 9E9, 9E9, 9E9]];
	VAR robtarget Openhole_2760 := [[400.77, -32.26, 175], [-0.112469, 0.698105, 0.680118, 0.193493], [0,0,0,0], [9E9, 9E9, 9E9, 9E9, 9E9, 9E9]];
	VAR robtarget Openhole_2761 := [[395.82, -31.65, 174.68], [-0.128411, 0.695349, 0.677033, 0.204026], [0,0,0,0], [9E9, 9E9, 9E9, 9E9, 9E9, 9E9]];
	VAR robtarget Openhole_2762 := [[394.83, -31.57, 174.6], [-0.131418, 0.694787, 0.676376, 0.206194], [0,0,0,0], [9E9, 9E9, 9E9, 9E9, 9E9, 9E9]];
